// TwinCAT 3 PLC project TwinCAT_OpenFramework_FileSystem
// Title: TwinCAT Open Framework File System
// Company: Oleksandr Tiutyk FOP
// Author: Oleksandr Tiutyk
// ProjectVersion: 1.0.13.0
// Description: TwinCAT.OpenFramework classes to work with files and directories
// ProgramVersion: 3.1.4026.28
// libraries:
//   Tc2_System, * (Beckhoff Automation GmbH)
//   Tc2_Utilities, * (Beckhoff Automation GmbH)
//   [TwinCAT Open Framework Core], * (Oleksandr Tiutyk FOP)
//   [TwinCAT Open Framework Tasks], * (Oleksandr Tiutyk FOP)
// project tree:
//   Exceptions/ IInvalidPathException.TcIO, InvalidPathException.TcPOU, IFileSystemException.TcIO, FileSystemException.TcPOU, FileSystemExceptions.TcPOU
//   Internal/ CurrentNamespace.TcPOU, NamespaceExtractor.TcPOU
//   / PathHelper.TcPOU
//   Tasks/Directory/ CreateDirectoryIfNotExists.TcPOU, CreateDirectory.TcPOU, RemoveEmptyDirectoryIfExists.TcPOU, RemoveEmptyDirectory.TcPOU, CheckDirectoryExists.TcPOU
//   Tasks/File/ DeleteFile.TcPOU, LoadFile.TcPOU, RenameFile.TcPOU
//   Tasks/File/FileContent/ FileContentManager.TcPOU, FileHandleResourceManager.TcPOU, FileHandleResource.TcPOU
//   Tasks/File/FileContent/Tasks/ CheckEndOfFile.TcPOU, FileContentTask.TcPOU, GetPositionInFile.TcPOU (not stored), IFileContentTask.TcIO, ReadBytesFromFile.TcPOU (not stored), ReadString255FromFile.TcPOU (not stored), SetPositionInFile.TcPOU, WriteBytesToFile.TcPOU, WriteString255ToFile.TcPOU (not stored)
//   Tasks/ IFileSystemTask.TcIO
//   Version/ Global_Version.TcGVL
// (motion and I/O tree: see PLC project twincat_openframework_core)
// real-time tasks:
//   TASK PlcTask: cycle T#10ms, priority 20, ADS port 350
//   TASK TestTask: cycle T#10ms, priority 1, ADS port 351
//   TASK RunnerTestTask: cycle T#10ms, priority 2, ADS port 354
//   TASK HowToTask: cycle T#10ms, priority 22, ADS port 353
// variable links:

// ---- Version/Global_Version.TcGVL
{attribute 'TcGenerated'}
{attribute 'no-analysis'}
{attribute 'linkalways'}
// This function has been automatically generated from the project information.
VAR_GLOBAL CONSTANT
	{attribute 'const_non_replaced'}
	stLibVersion_TwinCAT_Open_Framework_File_System : ST_LibVersion := (iMajor := 1, iMinor := 0, iBuild := 13, iRevision := 0, nFlags := 0, sVersion := '1.0.13.0');
END_VAR

// ---- Exceptions/IInvalidPathException.TcIO
(*
SPDX-FileCopyrightText: © 2026 Oleksandr Tiutyk <trofimich@gmail.com>
SPDX-License-Identifier: MIT
License: https://opensource.org/license/mit
*)

(*!
<summary>Exposes diagnostics for a rejected filesystem path.</summary>
<description>
Reports caller-detected path errors using the GeneralException lifetime and throw rules. The path is borrowed
during the call; errorMessage is copied by value.
</description>
*)
INTERFACE IInvalidPathException EXTENDS TOF_Core.IGeneralException

(*!
<summary>Raises an exception describing the rejected path and its reason.</summary>
<description>
Borrows path read-only for this call and copies errorMessage by value, limited to 255 characters. Retains
formatted diagnostic text, not the input reference. The caller detects the invalid path; this method does not
validate it.
</description>
*)
METHOD Throw
VAR_INPUT
	sourceNamespaceName : STRING;
	sourceClassName : STRING;
	sourcePOUName : STRING;
	sourcePosition : STRING;
END_VAR
VAR_IN_OUT CONSTANT
	path : STRING(255);
END_VAR
VAR_INPUT
	errorMessage : WSTRING(255);
END_VAR
END_METHOD

END_INTERFACE

// ---- Exceptions/IFileSystemException.TcIO
(*
SPDX-FileCopyrightText: © 2026 Oleksandr Tiutyk <trofimich@gmail.com>
SPDX-License-Identifier: MIT
License: https://opensource.org/license/mit
*)

(*!
<summary>Exposes diagnostics for a filesystem operation failure.</summary>
<description>
Reports caller-detected filesystem errors, such as ADS/OS errors, using the GeneralException lifetime and
throw rules. Message is borrowed read-only during the call; errorCode holds the operation failure code.
</description>
*)
INTERFACE IFileSystemException EXTENDS TOF_Core.IGeneralException

(*!
<summary>Raises an exception describing the filesystem failure.</summary>
<description>
Borrows message read-only for this call and records the numeric error code. Retains formatted diagnostic text.
The caller detects the filesystem error; this method propagates it.
</description>
<param name="sourceNamespaceName">Namespace of the caller.</param>
<param name="sourceClassName">Class name of the caller.</param>
<param name="sourcePOUName">POU name of the caller.</param>
<param name="sourcePosition">Source position of the caller.</param>
<param name="message">Diagnostic explanation.</param>
<param name="errorCode">Native/ADS error code, or 0 if unassigned.</param>
*)
METHOD Throw
VAR_INPUT
	sourceNamespaceName : STRING;
	sourceClassName : STRING;
	sourcePOUName : STRING;
	sourcePosition : STRING;
END_VAR
VAR_IN_OUT CONSTANT
	message : TOF_Core.ERROR_MESSAGE;
END_VAR
VAR_INPUT
	errorCode : UDINT := 0;
END_VAR
END_METHOD

END_INTERFACE

// ---- Tasks/File/FileContent/Tasks/IFileContentTask.TcIO
(*!
<summary>Defines a queued file operation that borrows a manager-owned resource.</summary>
<description>
A child must be READY and absent from every queue before binding. While queued, keep it alive and let the
queue drive its lifecycle. Binding and queue membership transfer no ownership. Implementations must keep
borrowed resource data read-only and complete pending I/O before permitting resource release. Keep the
resource owner alive throughout use. Removing a queue entry does not clear the binding.
</description>
*)
INTERFACE IFileContentTask EXTENDS IFileSystemTask

(*!
<summary>Provides the native handle associated with the file resource.</summary>
<description>
Use only during the current acquisition; the value alone is not an acquisition guard. Do not close it
independently or retain it across release. FileContentTask returns zero when unbound.
</description>
*)
{attribute 'monitoring' := 'call'}
PROPERTY FileHandle : UINT
GET
END_GET
END_PROPERTY

(*!
<summary>Provides a copy of the path from the borrowed file resource.</summary>
<description>
The resource owner must remain alive during access. FileContentTask returns an empty string when unbound. The
path is configuration, not proof of acquisition or file existence.
</description>
*)
{attribute 'monitoring' := 'call'}
PROPERTY FINAL FilePath : Tc2_System.T_MaxString
GET
END_GET
END_PROPERTY

(*!
<summary>Bind, replace or clear a borrowed resource only in READY; otherwise throw.</summary>
<description>
An invalid reference clears the binding. Reset a STOPPED task before rebinding. The caller must first remove
the task from any queue; READY alone does not mean it is unqueued. The resource owner must outlive its use by
this task. FileContentTask clears binding on Reset from STOPPED, but its READY Reset is a no-op; a removed
READY child needs explicit clearing or rebinding.
</description>
*)

METHOD SetFileHandleResource
VAR_INPUT
	fileHandleResource : REFERENCE TO FileHandleResource;
END_VAR
END_METHOD

END_INTERFACE

// ---- Tasks/IFileSystemTask.TcIO
(*!
<summary>Provides task execution with a configured file-system target and operation timeout.</summary>
<description>
Before online change, the application must stop submitting new work and keep advancing each running task
through completion and cleanup. Keep its configuration, borrowed objects and buffers alive until then. Drive
queued children only through their owning queue. File-content tasks also require their resource owner to
finish release; a stopped child alone does not close its file. Online change with pending native operations or
retained open resources is unsupported. This is an application precondition, not an automatic online-change
guard. Completed best-effort cleanup does not certify physical resource release after a native close or
enumeration-abort failure.
</description>
*)
INTERFACE IFileSystemTask EXTENDS TOF_Tasks.ITask

(*!
<summary>Selects the ADS target for the native filesystem operation.</summary>
<description>
Configure before execution and keep stable through stopping. File-content tasks obtain the effective target
from their bound resource; assigning this property does not retarget an acquired file.
</description>
*)
{attribute 'monitoring' := 'call'}
PROPERTY AmsNetId : Tc2_System.T_AmsNetID
GET
END_GET
SET
END_SET
END_PROPERTY

(*!
<summary>Configures the timeout passed to native operation requests.</summary>
<description>
Implementations apply this value to their native requests. Configure before execution and keep stable through
stopping; it is not a deadline for the entire task lifecycle.
</description>
*)
{attribute 'monitoring' := 'call'}
PROPERTY Timeout : TIME
GET
END_GET
SET
END_SET
END_PROPERTY

END_INTERFACE

// ---- Exceptions/InvalidPathException.TcPOU
(*
SPDX-FileCopyrightText: © 2026 Oleksandr Tiutyk <trofimich@gmail.com>
SPDX-License-Identifier: MIT
License: https://opensource.org/license/mit
*)

(*!
<summary>Reports a rejected filesystem path and its diagnostic explanation.</summary>
<description>
Reports caller-detected path errors using the GeneralException lifetime and throw rules. The path is borrowed
during the call; errorMessage is copied by value. Dynamic copies are explicitly registered by Clone after
construction; plain __NEW does not transfer ownership to the task manager.
</description>
*)

{attribute 'enable_dynamic_creation'}
{attribute 'no_explicit_call' := 'do not call this function block directly'}
FUNCTION_BLOCK InvalidPathException EXTENDS TOF_Core.GeneralException IMPLEMENTS IInvalidPathException
VAR_STAT
	//! <summary>Class name shared by all instances of this function block.</summary>
	{attribute 'hide'} 
	_ClassName : STRING := __POUNAME();
END_VAR

(*!
<summary>Provides the concrete type name used in diagnostics.</summary>
<description>
Returns borrowed read-only metadata; keep the instance alive and do not modify the referenced string.
Reading does not allocate memory, initialize resources or transfer ownership.
</description>
*)
{attribute 'monitoring' := 'call'}
PROPERTY ClassName : REFERENCE TO STRING
GET
ClassName REF= _ClassName;
END_GET
END_PROPERTY

(*!
<summary>Creates a task-owned copy of this exception and its diagnostic payload.</summary>
<description>
Registers the newly constructed instance before copying payload, outside FB_init. Registration failure
releases the unregistered instance and raises a terminal error; copy failure leaves the registered instance
owned by the task manager for cleanup. Custom overrides must follow the same ownership sequence. The returned
reference is borrowed until task cleanup and must not be deleted by the caller.
</description>
*)
METHOD Clone : TOF_Core.IObject
VAR
	exceptionClone : POINTER TO InvalidPathException;
END_VAR
exceptionClone := __NEW(InvalidPathException);

IF exceptionClone = 0 THEN
	TOF_Core.DynamicMemoryManager.RaiseAllocationFailure();
END_IF

TOF_Core.DynamicMemoryManager.RegisterAutoDisposedObject(autoDisposedObject := exceptionClone^);

exceptionClone^.CopyGeneralFields(sourceException := THIS^);

Clone := exceptionClone^;
END_METHOD

(*!
<summary>Provides the library namespace used in diagnostics.</summary>
<description>Returns borrowed read-only namespace storage; do not modify the referenced string.</description>
*)
{attribute 'monitoring' := 'call'}
PROPERTY NamespaceName : REFERENCE TO STRING
GET
NamespaceName REF= CurrentNamespace.Name;
END_GET
END_PROPERTY

(*!
<summary>Reports the size of this concrete instance in bytes.</summary>
*)
{attribute 'monitoring' := 'call'}
PROPERTY SelfSize : ULINT
GET
SelfSize := XSIZEOF(THIS^);
END_GET
END_PROPERTY

(*!
<summary>Raises an exception describing the rejected path and its reason.</summary>
<description>
Borrows path read-only for this call and copies errorMessage by value, limited to 255 characters. Formats
diagnostic text without heap allocation during message preparation; does not retain the input reference. The
caller detects the invalid path; this method does not validate it.
</description>
*)
METHOD Throw
VAR_INPUT
	sourceNamespaceName : STRING;
	sourceClassName : STRING;
	sourcePOUName : STRING;
	sourcePosition : STRING;
END_VAR
VAR_IN_OUT CONSTANT
	path : STRING(255);
END_VAR
VAR_INPUT
	errorMessage : WSTRING(255);
END_VAR
VAR
	message : TOF_Core.ERROR_MESSAGE;
END_VAR
TOF_Core.WideStrings.Append255(
	message,
	"Invalid path ",
	TO_WSTRING('$22'),
	TO_WSTRING(path),
	TO_WSTRING('$22: '),
	errorMessage);

InternalThrow(
	sourceNamespaceName := sourceNamespaceName,
	sourceClassName := sourceClassName,
	sourcePOUName := sourcePOUName,
	sourcePosition := sourcePosition,
	message := message,
	errorCode := 0,
	innerException := 0
);
END_METHOD

END_FUNCTION_BLOCK

// ---- Internal/CurrentNamespace.TcPOU
(*
SPDX-FileCopyrightText: © 2026 Oleksandr Tiutyk <trofimich@gmail.com>
SPDX-License-Identifier: MIT
License: https://opensource.org/license/mit
*)

(*!
<summary>Owns the namespace storage shared by FileSystem diagnostic metadata.</summary>
*)

{attribute 'no_explicit_call' := 'do not call this POU directly'}
PROGRAM INTERNAL CurrentNamespace
VAR
	{attribute 'hide'} 
	_NamespaceExtractor : NamespaceExtractor;
END_VAR

(*!
<summary>Provides the compiler-initialized namespace string for this library.</summary>
<description>Returns borrowed read-only storage owned by the internal namespace extractor.</description>
*)
{attribute 'monitoring' := 'call'}
PROPERTY Name : REFERENCE TO STRING
GET
Name REF= _NamespaceExtractor.CurrentNamespace;
END_GET
END_PROPERTY

END_PROGRAM

// ---- Internal/NamespaceExtractor.TcPOU
(*
SPDX-FileCopyrightText: © 2026 Oleksandr Tiutyk <trofimich@gmail.com>
SPDX-License-Identifier: MIT
License: https://opensource.org/license/mit
*)

(*!
<summary>Receives the library namespace through compiler initialization.</summary>
<description>
CurrentNamespace is metadata storage; callers borrow it read-only through CurrentNamespace.Name.
</description>
*)

FUNCTION_BLOCK INTERNAL NamespaceExtractor
VAR_OUTPUT
	{attribute 'init_namespace'} 
	CurrentNamespace : STRING; 	
END_VAR

END_FUNCTION_BLOCK

// ---- Exceptions/FileSystemException.TcPOU
(*
SPDX-FileCopyrightText: © 2026 Oleksandr Tiutyk <trofimich@gmail.com>
SPDX-License-Identifier: MIT
License: https://opensource.org/license/mit
*)

(*!
<summary>Reports an error occurring during filesystem operations.</summary>
<description>
Reports caller-detected filesystem failures using the GeneralException lifetime and throw rules. Message is
borrowed read-only during the call; errorCode stores the native/ADS error identifier. Dynamic instances and
clones belong to DynamicMemoryManager until task cleanup. Plain __NEW does not transfer ownership to the task
manager.
</description>
*)

{attribute 'enable_dynamic_creation'}
{attribute 'no_explicit_call' := 'do not call this function block directly'}
FUNCTION_BLOCK FileSystemException EXTENDS TOF_Core.GeneralException IMPLEMENTS IFileSystemException
VAR_STAT
	{attribute 'hide'} 
	_ClassName : STRING := __POUNAME();
END_VAR

(*!
<summary>Provides the concrete type name used in diagnostics.</summary>
<description>
Returns borrowed read-only metadata; keep the instance alive and do not modify the referenced string.
Reading does not allocate memory, initialize resources or transfer ownership.
</description>
*)
{attribute 'monitoring' := 'call'}
PROPERTY ClassName : REFERENCE TO STRING
GET
ClassName REF= _ClassName;
END_GET
END_PROPERTY

(*!
<summary>Creates a task-owned copy of this exception and its diagnostic payload.</summary>
<description>
Registers the newly constructed instance before copying payload, outside FB_init. Registration failure
releases the unregistered instance and raises a terminal error; copy failure leaves the registered instance
owned by the task manager for cleanup. Custom overrides must follow the same ownership sequence. The returned
reference is borrowed until task cleanup and must not be deleted by the caller.
</description>
*)
METHOD Clone : TOF_Core.IObject
VAR
	exceptionClone : POINTER TO FileSystemException;
END_VAR
exceptionClone := __NEW(FileSystemException);

IF exceptionClone = 0 THEN
	TOF_Core.DynamicMemoryManager.RaiseAllocationFailure();
END_IF

TOF_Core.DynamicMemoryManager.RegisterAutoDisposedObject(autoDisposedObject := exceptionClone^);

exceptionClone^.CopyGeneralFields(sourceException := THIS^);

Clone := exceptionClone^;
END_METHOD

(*!
<summary>Provides the library namespace used in diagnostics.</summary>
<description>Returns borrowed read-only namespace storage; do not modify the referenced string.</description>
*)
{attribute 'monitoring' := 'call'}
PROPERTY NamespaceName : REFERENCE TO STRING
GET
NamespaceName REF= CurrentNamespace.Name;
END_GET
END_PROPERTY

(*!
<summary>Reports the size of this concrete instance in bytes.</summary>
*)
{attribute 'monitoring' := 'call'}
PROPERTY SelfSize : ULINT
GET
SelfSize := XSIZEOF(THIS^);
END_GET
END_PROPERTY

(*!
<summary>Raises a filesystem exception with the supplied message and error code.</summary>
<description>
Borrows message read-only for this call and records the numeric error code. Formats diagnostic text without
heap allocation during message preparation; does not retain the input reference. The caller detects the
filesystem error; this method propagates it.
</description>
<param name="sourceNamespaceName">Namespace of the caller.</param>
<param name="sourceClassName">Class name of the caller.</param>
<param name="sourcePOUName">POU name of the caller.</param>
<param name="sourcePosition">Source position of the caller.</param>
<param name="message">Diagnostic explanation.</param>
<param name="errorCode">Native/ADS error code, or 0 if unassigned.</param>
*)
METHOD Throw
VAR_INPUT
	sourceNamespaceName : STRING;
	sourceClassName : STRING;
	sourcePOUName : STRING;
	sourcePosition : STRING;
END_VAR
VAR_IN_OUT CONSTANT
	message : TOF_Core.ERROR_MESSAGE;
END_VAR
VAR_INPUT
	errorCode : UDINT := 0;
END_VAR
InternalThrow(
	sourceNamespaceName := sourceNamespaceName,
	sourceClassName := sourceClassName,
	sourcePOUName := sourcePOUName,
	sourcePosition := sourcePosition,
	message := message,
	errorCode := errorCode,
	innerException := 0
);
END_METHOD

END_FUNCTION_BLOCK

// ---- Exceptions/FileSystemExceptions.TcPOU
(*
SPDX-FileCopyrightText: © 2026 Oleksandr Tiutyk <trofimich@gmail.com>
SPDX-License-Identifier: MIT
License: https://opensource.org/license/mit
*)

(*!
<summary>Provides static helper methods for throwing FileSystem-specific exceptions.</summary>
<description>
Constructs stack-local template exceptions, formats diagnostics without heap allocation and propagates them
through ExceptionManager.
</description>
*)

PROGRAM FileSystemExceptions
VAR
	{attribute 'hide'} 
	_ClassName : STRING := __POUNAME();
END_VAR

//! <summary>Borrows the concrete class name for the lifetime of this instance; callers must not modify it.</summary>
{attribute 'monitoring' := 'call'}
PROPERTY ClassName : REFERENCE TO STRING
GET
ClassName REF= _ClassName;
END_GET
END_PROPERTY

//! <summary>Borrows the compiler-initialized namespace; callers must not modify the returned reference.</summary>
{attribute 'monitoring' := 'call'}
PROPERTY NamespaceName : REFERENCE TO STRING
GET
NamespaceName REF= CurrentNamespace.Name;
END_GET
END_PROPERTY

(*!
<summary>Raises a FileSystemException without requiring a caller-owned exception variable.</summary>
<description>Constructs a temporary stack template and delegates to FileSystemException.Throw.</description>
<param name="sourceNamespaceName">Namespace of the caller.</param>
<param name="sourceClassName">Class name of the caller.</param>
<param name="sourcePOUName">POU name of the caller.</param>
<param name="sourcePosition">Source position of the caller.</param>
<param name="message">Diagnostic explanation.</param>
<param name="errorCode">Native/ADS error code, or 0 if unassigned.</param>
*)
METHOD ThrowFileSystem
VAR_INPUT
	sourceNamespaceName : STRING;
	sourceClassName : STRING;
	sourcePOUName : STRING;
	sourcePosition : STRING;
END_VAR
VAR_IN_OUT CONSTANT
	message : TOF_Core.ERROR_MESSAGE;
END_VAR
VAR_INPUT
	errorCode : UDINT := 0;
END_VAR
VAR
	exception : FileSystemException;
END_VAR
exception.Throw(
	sourceNamespaceName := sourceNamespaceName,
	sourceClassName := sourceClassName,
	sourcePOUName := sourcePOUName,
	sourcePosition := sourcePosition,
	message := message,
	errorCode := errorCode
);
END_METHOD

(*!
<summary>Raises an InvalidPathException without requiring a caller-owned exception variable.</summary>
<description>Constructs a temporary stack template and delegates to InvalidPathException.Throw.</description>
<param name="sourceNamespaceName">Namespace of the caller.</param>
<param name="sourceClassName">Class name of the caller.</param>
<param name="sourcePOUName">POU name of the caller.</param>
<param name="sourcePosition">Source position of the caller.</param>
<param name="path">Rejected filesystem path.</param>
<param name="errorMessage">Diagnostic explanation.</param>
*)
METHOD ThrowInvalidPath
VAR_INPUT
	sourceNamespaceName : STRING;
	sourceClassName : STRING;
	sourcePOUName : STRING;
	sourcePosition : STRING;
END_VAR
VAR_IN_OUT CONSTANT
	path : STRING(255);
END_VAR
VAR_INPUT
	errorMessage : WSTRING(255);
END_VAR
VAR
	exception : InvalidPathException;
END_VAR
exception.Throw(
	sourceNamespaceName := sourceNamespaceName,
	sourceClassName := sourceClassName,
	sourcePOUName := sourcePOUName,
	sourcePosition := sourcePosition,
	path := path,
	errorMessage := errorMessage
);
END_METHOD

END_PROGRAM

// ---- PathHelper.TcPOU
(*
SPDX-FileCopyrightText: © 2026 Oleksandr Tiutyk <trofimich@gmail.com>
SPDX-License-Identifier: MIT
License: https://opensource.org/license/mit
*)

(*!
<summary>Provides lexical checks for directory and file path strings.</summary>
<description>
These checks perform no filesystem I/O, normalization or access checks. Passing does not certify acceptance by
a native service or target filesystem. The current filter is not a complete Windows, UNC or platform-specific
path validator; it does not validate reserved names or dot components. Callers must separately satisfy the
path requirements of the actual operation and target.
</description>
*)

{attribute 'no_explicit_call' := 'do not call this function block directly'}
PROGRAM PathHelper
VAR CONSTANT
	//! <summary>Drive-letter, colon and separator occupy the first three bytes of an absolute drive prefix.</summary>
	_DrivePrefixLength : UDINT := 3;
	//! <summary>Zero-based index of the colon immediately following a drive letter.</summary>
	_DriveColonIndex : UDINT := 1;
	//! <summary>Zero-based index of the separator following the drive colon.</summary>
	_DriveSeparatorIndex : UDINT := 2;
	//! <summary>Last index allowed in the initial separator pair before repeated separators are rejected.</summary>
	_LeadingSeparatorPairLastIndex : UDINT := 1;
END_VAR
VAR
	{attribute 'hide'} 
	_ClassName : STRING := __POUNAME();
END_VAR

//! <summary>Borrows the concrete class name for the lifetime of this instance; callers must not modify it.</summary>
{attribute 'monitoring' := 'call'}
PROPERTY ClassName : REFERENCE TO STRING
GET
ClassName REF= _ClassName;
END_GET
END_PROPERTY

(*!
<summary>Checks the lexical form of a directory path without accessing the filesystem.</summary>
<description>
Rejects an empty path, bytes below ASCII space, characters from the current forbidden set and repeated
slash/backslash separators beyond the leading pair. A colon is accepted only immediately after an ASCII drive
letter and before a separator. Relative paths and a trailing separator are not rejected solely for being
relative or trailing. Leading separator pairs are permitted lexically, but UNC server/share structure is not
checked and native network-path support is not implied. Reserved names, dot components and trailing
dots/spaces are not validated. TRUE means only that this filter passed; errorMessage is meaningful on FALSE.
Input is borrowed only for the call.
</description>
<param name="directoryPath">Directory path to inspect without modifying or retaining it.</param>
<param name="errorMessage">Reason for the first rejected condition.</param>
*)
METHOD IsValidDirectoryPath : BOOL
VAR_IN_OUT CONSTANT
	directoryPath : Tc2_System.T_MaxString;
END_VAR
VAR_OUTPUT
	errorMessage : WSTRING(255);
END_VAR
VAR
	i, j : UDINT;
	stringLength : UDINT;
	character : BYTE;

	(* Current lexical exclusions, not an OS-wide list. Caret is an existing library restriction;
	   the drive-letter exception below handles the only accepted colon position. *)
	invalidChars : STRING(8) := '<>"|?*^:';
END_VAR
stringLength := TOF_Core.Strings.GetLength(value := directoryPath);

IF stringLength = TOF_Core.UnsignedInt32.ZERO THEN
	errorMessage := "Path is empty";
	RETURN;
END_IF

FOR i := 0 TO stringLength - 1 DO
	character := directoryPath[i];

	(* A colon is allowed only in an absolute ASCII drive prefix. *)
	IF i = _DriveColonIndex AND_THEN character = Tc2_System.F_ToASC(str := ':') THEN

		IF stringLength >= _DrivePrefixLength
			AND_THEN (
				directoryPath[_DriveSeparatorIndex] = Tc2_System.F_ToASC(str := '\')
				OR_ELSE directoryPath[_DriveSeparatorIndex] = Tc2_System.F_ToASC(str := '/')
			)
			AND_THEN (
				(directoryPath[0] >= Tc2_System.F_ToASC(str := 'A')
					AND_THEN directoryPath[0] <= Tc2_System.F_ToASC(str := 'Z'))
				OR_ELSE (directoryPath[0] >= Tc2_System.F_ToASC(str := 'a')
					AND_THEN directoryPath[0] <= Tc2_System.F_ToASC(str := 'z'))
			)
		THEN
			CONTINUE;
		END_IF

	END_IF

	FOR j := 0 TO TOF_Core.Strings.GetLength(value := invalidChars) - 1 DO

		IF character = invalidChars[j] THEN
			errorMessage := TOF_Core.WideStrings.Concat255(
				"The forbidden character '",
				TO_WSTRING(Tc2_System.F_ToCHR(c := character)),
				"' at position ",
				TO_WSTRING(i + 1)
			);
			RETURN;
		END_IF

	END_FOR

	IF character < TOF_Core.Strings.ASCII_SPACE THEN
		errorMessage := TOF_Core.WideStrings.Concat255(
			"The forbidden character with code ",
			TO_WSTRING(character),
			" at position ",
			TO_WSTRING(i + 1)
		);
		RETURN;
	END_IF

	IF i > _LeadingSeparatorPairLastIndex
		AND_THEN (character = Tc2_System.F_ToASC(str := '\') OR_ELSE character = Tc2_System.F_ToASC(str := '/'))
		AND_THEN (
			directoryPath[i - 1] = Tc2_System.F_ToASC(str := '\')
			OR_ELSE directoryPath[i - 1] = Tc2_System.F_ToASC(str := '/')
		)
	THEN
		errorMessage := TOF_Core.WideStrings.Concat255("Several slashes one by one at position ", TO_WSTRING(i + 1));
		RETURN;
	END_IF

END_FOR

IsValidDirectoryPath := TRUE;
END_METHOD

(*!
<summary>Checks the lexical form of a file path and rejects a trailing separator.</summary>
<description>
Borrows the path only for this call. Returns FALSE with errorMessage for an empty path, a forbidden character,
repeated separators beyond the leading pair, or a final slash or backslash. A drive-letter colon is allowed
only before a slash or backslash. TRUE means the lexical checks passed; it does not establish file existence,
access rights or acceptance by the target filesystem. No filesystem I/O is performed. Relative paths are not
rejected solely for being relative. Leading separator pairs do not establish a valid UNC path; reserved names,
dot components and trailing dots/spaces are not validated. errorMessage is meaningful only when FALSE is
returned.
</description>
<param name="filePath">File path to inspect without modifying or retaining it.</param>
<param name="errorMessage">Receives the reason for the first rejected condition.</param>
*)
METHOD IsValidFilePath : BOOL
VAR_IN_OUT CONSTANT
	filePath : Tc2_System.T_MaxString;
END_VAR
VAR_OUTPUT
	errorMessage : WSTRING(255);
END_VAR
VAR
	i, j : UDINT;
	stringLength : UDINT;
	character : BYTE;

	(* Current lexical exclusions, not an OS-wide list. Caret is an existing library restriction;
	   the drive-letter exception below handles the only accepted colon position. *)
	invalidChars : STRING(8) := '<>"|?*^:';
END_VAR
stringLength := TOF_Core.Strings.GetLength(value := filePath);

IF stringLength = TOF_Core.UnsignedInt32.ZERO THEN
	errorMessage := "Path is empty";
	RETURN;
END_IF

FOR i := 0 TO stringLength - 1 DO
	character := filePath[i];

	(* A colon is allowed only in an absolute ASCII drive prefix. *)
	IF i = _DriveColonIndex AND_THEN character = Tc2_System.F_ToASC(str := ':') THEN

		IF stringLength >= _DrivePrefixLength
			AND_THEN (
				filePath[_DriveSeparatorIndex] = Tc2_System.F_ToASC(str := '\')
				OR_ELSE filePath[_DriveSeparatorIndex] = Tc2_System.F_ToASC(str := '/')
			)
			AND_THEN (
				(filePath[0] >= Tc2_System.F_ToASC(str := 'A')
					AND_THEN filePath[0] <= Tc2_System.F_ToASC(str := 'Z'))
				OR_ELSE (filePath[0] >= Tc2_System.F_ToASC(str := 'a')
					AND_THEN filePath[0] <= Tc2_System.F_ToASC(str := 'z'))
			)
		THEN
			CONTINUE;
		END_IF

	END_IF

	FOR j := 0 TO TOF_Core.Strings.GetLength(value := invalidChars) - 1 DO

		IF character = invalidChars[j] THEN
			errorMessage := TOF_Core.WideStrings.Concat255(
				"The forbidden character '",
				TO_WSTRING(Tc2_System.F_ToCHR(c := character)),
				"' at position ",
				TO_WSTRING(i + 1)
			);
			RETURN;
		END_IF

	END_FOR

	IF character < TOF_Core.Strings.ASCII_SPACE THEN
		errorMessage := TOF_Core.WideStrings.Concat255(
			"The forbidden character with code ",
			TO_WSTRING(character),
			" at position ",
			TO_WSTRING(i + 1)
		);
		RETURN;
	END_IF

	IF i > _LeadingSeparatorPairLastIndex
		AND_THEN (character = Tc2_System.F_ToASC(str := '\') OR_ELSE character = Tc2_System.F_ToASC(str := '/'))
		AND_THEN (
			filePath[i - 1] = Tc2_System.F_ToASC(str := '\')
			OR_ELSE filePath[i - 1] = Tc2_System.F_ToASC(str := '/')
		)
	THEN
		errorMessage := TOF_Core.WideStrings.Concat255("Several slashes one by one at position ", TO_WSTRING(i + 1));
		RETURN;
	END_IF

	IF i = stringLength - 1
		AND_THEN (character = Tc2_System.F_ToASC(str := '\') OR_ELSE character = Tc2_System.F_ToASC(str := '/'))
	THEN
		errorMessage := "Slash at the end of the path";
		RETURN;
	END_IF

END_FOR

IsValidFilePath := TRUE;
END_METHOD

//! <summary>Borrows the compiler-initialized namespace; callers must not modify the returned reference.</summary>
{attribute 'monitoring' := 'call'}
PROPERTY NamespaceName : REFERENCE TO STRING
GET
NamespaceName REF= CurrentNamespace.Name;
END_GET
END_PROPERTY

END_PROGRAM

// ---- Tasks/Directory/CreateDirectoryIfNotExists.TcPOU
(*
SPDX-FileCopyrightText: © 2026 Oleksandr Tiutyk <trofimich@gmail.com>
SPDX-License-Identifier: MIT
License: https://opensource.org/license/mit
*)

(*!
<summary>Creates a filesystem directory when it is absent.</summary>
<description>
An existing directory completes after native enumeration has been closed. Pending search and create commands
finish before stopping. Diagnostic string inputs are borrowed only during the call; retained diagnostic text
is copied into owned storage. A found file produces FAILURE without starting create I/O; stopping closes the
enumeration before task completion. The existence check and subsequent filesystem change are separate,
non-atomic operations. Another actor may change the same path between them. Native errors from the subsequent
create/remove are reported as failure; this wrapper does not retry or reinterpret them as a successful race.
Coordinate access externally when other tasks or processes can modify the same path. Cancellation does not
roll back completed filesystem effects.
</description>
*)

{attribute 'no_explicit_call' := 'do not call this function block directly'}
FUNCTION_BLOCK CreateDirectoryIfNotExists EXTENDS TOF_Tasks.Task IMPLEMENTS IFileSystemTask
VAR_STAT
	//! <summary>Static type metadata available before the base task initializes its default name.</summary>
	{attribute 'hide'}
	_ClassName : STRING := __POUNAME();
END_VAR
VAR
	_DirectoryChecking : BOOL;

	_EnumFindFile : Tc2_Utilities.FB_EnumFindFileEntry;
	//! <summary>Records whether a search command may still own native enumeration resources.</summary>
	_EnumerationStarted : BOOL;
	//! <summary>Prevents repeating the abort command while its completion is pending.</summary>
	_EnumerationAbortIssued : BOOL;

    _CreateDirectory : Tc2_System.FB_CreateDir;
END_VAR

(*!
<summary>Selects the ADS target for the native filesystem operation.</summary>
<description>
Configure before Start and keep unchanged until STOPPED; the setter stores configuration without submitting
I/O.
</description>
*)
{attribute 'monitoring' := 'call'}
PROPERTY AmsNetId : Tc2_System.T_AmsNetID
GET
AmsNetId := _CreateDirectory.sNetId;
END_GET
SET
_CreateDirectory.sNetId := AmsNetId;
_EnumFindFile.sNetId := AmsNetId;
END_SET
END_PROPERTY

(*!
<summary>Provides the concrete type name used in diagnostics.</summary>
<description>
Returns borrowed read-only metadata; keep the instance alive and do not modify the referenced string.
Initialized static storage is ready during base Task.FB_init; this getter has no side effects or exceptions.
</description>
*)
{attribute 'monitoring' := 'call'}
PROPERTY ClassName : REFERENCE TO STRING
GET
ClassName REF= _ClassName;
END_GET
END_PROPERTY

(*!
<summary>Provides the copied directory path used by the operation and its existence check.</summary>
<description>
Configure before Start and keep unchanged until STOPPED. PathHelper applies its limited lexical filter before
native submission. Assignment does not perform I/O; Reset preserves the path.
</description>
*)
{attribute 'monitoring' := 'call'}
PROPERTY DirectoryPath : Tc2_System.T_MaxString
GET
DirectoryPath := _CreateDirectory.sPathName;
END_GET
SET
_CreateDirectory.sPathName := DirectoryPath;
_EnumFindFile.sPathName := DirectoryPath;
END_SET
END_PROPERTY

(*!
<summary>Provides the library namespace used in diagnostics.</summary>
<description>Returns borrowed read-only namespace storage; do not modify the referenced string.</description>
*)
{attribute 'monitoring' := 'call'}
PROPERTY NamespaceName : REFERENCE TO STRING
GET
NamespaceName REF= CurrentNamespace.Name;
END_GET
END_PROPERTY

(*!
<summary>Clears completed directory operations and per-run enumeration cleanup state.</summary>
<description>Called only after stopping has completed; it does not abandon pending native I/O.</description>
*)
METHOD PROTECTED OnReset
_EnumFindFile(bExecute := FALSE);
_CreateDirectory(bExecute := FALSE);

_DirectoryChecking := FALSE;
_EnumerationStarted := FALSE;
_EnumerationAbortIssued := FALSE;
END_METHOD

(*!
<summary>Checks for a directory and creates it only if absent.</summary>
<description>
Early discovery leaves native search cleanup to OnStopping. A missing directory begins a create request after
bEOE. Computed diagnostics are held in local buffers for the receiving call without dynamic string-builder
allocations. A found file returns ERROR with a diagnostic message and leaves enumeration cleanup to
OnStopping; no create request starts.
</description>
<param name="processingState">
BUSY while searching or creating; DONE when no create is needed or creation ends; ERROR when the path refers
to a file.
</param>
<param name="stopReasonMessage">
Receives diagnostics when the path refers to a file; native failures use exceptions.
</param>
*)
METHOD PROTECTED OnRunning
VAR_OUTPUT
	processingState : TOF_Tasks.TASK_PROCESSING_STATE;
END_VAR
VAR_IN_OUT
	stopReasonMessage : TOF_Core.ERROR_MESSAGE;
END_VAR
VAR
	formattedExceptionMessage : TOF_Core.ERROR_MESSAGE;
	pathErrorMessage : WSTRING(255);
END_VAR
IF NOT _EnumFindFile.bExecute THEN 
	IF TOF_Core.Strings.IsNullOrWhiteSpace(stringToCheck := _EnumFindFile.sPathName) THEN
		TOF_Core.Exceptions.ThrowDataMemberNotSpecified(
			sourceNamespaceName := NamespaceName,
			sourceClassName := ClassName,
			sourcePOUName := __POUNAME(),
			sourcePosition := __POSITION(),
			dataMemberName := 'DirectoryPath'
		);		
	END_IF
	
	IF NOT PathHelper.IsValidDirectoryPath(directoryPath := _EnumFindFile.sPathName, errorMessage => pathErrorMessage) THEN
		FileSystemExceptions.ThrowInvalidPath(
			sourceNamespaceName := NamespaceName,
			sourceClassName := ClassName,
			sourcePOUName := __POUNAME(),
			sourcePosition := __POSITION(),
			path := _EnumFindFile.sPathName,
			errorMessage := pathErrorMessage
		);
	END_IF
	
	_DirectoryChecking := TRUE;
	
	_EnumFindFile.eCmd := Tc2_Utilities.E_EnumCmdType.eEnumCmd_First;
END_IF

IF _DirectoryChecking THEN
	_EnumerationStarted := TRUE;
	_EnumFindFile(bExecute := TRUE);
	
	IF _EnumFindFile.bError THEN
		TOF_Core.WideStrings.Append255(
			formattedExceptionMessage,
			"Error while checking directory '",
			TO_WSTRING(_EnumFindFile.sPathName),
			"'");

		FileSystemExceptions.ThrowFileSystem(
			sourceNamespaceName := NamespaceName,
			sourceClassName := ClassName,
			sourcePOUName := __POUNAME(),
			sourcePosition := __POSITION(),
			message := formattedExceptionMessage,
			errorCode := _EnumFindFile.nErrId
		);
	ELSIF NOT _EnumFindFile.bBusy THEN	
		_DirectoryChecking := FALSE;
		
		IF NOT _EnumFindFile.bEOE THEN
			IF _EnumFindFile.stFindFile.fileAttributes.bDirectory THEN
				processingState := TOF_Tasks.TASK_PROCESSING_STATE.DONE;
			ELSE
				stopReasonMessage := TOF_Core.WideStrings.Concat255("Directory path refers to a file: ", TO_WSTRING(_EnumFindFile.sPathName));
				processingState := TOF_Tasks.TASK_PROCESSING_STATE.ERROR;
			END_IF
		END_IF
	END_IF
ELSE
	_CreateDirectory(bExecute := TRUE);
	
	IF _CreateDirectory.bError THEN
		TOF_Core.WideStrings.Append255(
			formattedExceptionMessage,
			"Error while creating directory '",
			TO_WSTRING(_CreateDirectory.sPathName),
			"'");

		FileSystemExceptions.ThrowFileSystem(
			sourceNamespaceName := NamespaceName,
			sourceClassName := ClassName,
			sourcePOUName := __POUNAME(),
			sourcePosition := __POSITION(),
			message := formattedExceptionMessage,
			errorCode := _CreateDirectory.nErrId
		);
	END_IF
	
	IF NOT _CreateDirectory.bBusy THEN
		processingState := TOF_Tasks.TASK_PROCESSING_STATE.DONE;
	END_IF	
END_IF
END_METHOD

(*!
<summary>Advances directory stop actions before reporting termination.</summary>
<description>
Used for every stop reason. Drains a pending search, then issues an abort with a rising bExecute edge if the
search ended before bEOE without error. Waits for abort and any pending create operation before termination;
no new ordinary create request starts. An abort error is logged once with its native code and path, without
retrying abort or replacing the task stop reason. Readiness means this cleanup attempt ended, not that server
resources were proven released. The log attempt is made after clearing pending enumeration state; logger
failure does not restart cleanup.
</description>
<param name="readyToRelease">TRUE when the directory FBs have finished their pending requests.</param>
*)
METHOD PROTECTED OnStopping
VAR_OUTPUT
	readyToRelease : BOOL;
END_VAR
VAR
	enumerationAbortMessage : WSTRING(255);
END_VAR
IF _EnumerationStarted THEN
	_EnumFindFile(bExecute := FALSE);

	IF NOT _EnumFindFile.bBusy THEN

		IF _EnumFindFile.bEOE OR_ELSE _EnumFindFile.bError THEN
			_EnumerationStarted := FALSE;

			(* End this attempt before reporting its error so logging cannot cause repeated aborts. *)

			IF _EnumerationAbortIssued AND_THEN _EnumFindFile.bError THEN
				enumerationAbortMessage := TOF_Core.WideStrings.Concat255(
					"Directory enumeration abort failed (native error code ",
					TO_WSTRING(_EnumFindFile.nErrId),
					"): ",
					TO_WSTRING(_EnumFindFile.sPathName)
				);
				TryLogDiagnosticMessage(
					message := enumerationAbortMessage,
					category := TOF_Core.LOG_CATEGORY.ERROR,
					topic1 := TO_WSTRING(__POUNAME())
				);
			END_IF

		ELSIF NOT _EnumerationAbortIssued THEN
			_EnumFindFile(bExecute := TRUE, eCmd := Tc2_Utilities.E_EnumCmdType.eEnumCmd_Abort);
			_EnumerationAbortIssued := TRUE;
		ELSE
			_EnumerationStarted := FALSE;
		END_IF

	END_IF

END_IF

_CreateDirectory(bExecute := FALSE);

readyToRelease := NOT _EnumerationStarted AND_THEN NOT _CreateDirectory.bBusy;
END_METHOD

(*!
<summary>Selects the native path context for the filesystem request.</summary>
<description>
Configure before Start and keep unchanged until STOPPED. It is passed to the native operation, not used as a
path-validity result. Reset preserves it. Target support includes the ePath enumeration input in
Tc2_Utilities 3.10.9.
</description>
*)
{attribute 'monitoring' := 'call'}
PROPERTY PathType : Tc2_System.E_OpenPath
GET
PathType := _CreateDirectory.ePath;
END_GET
SET
_CreateDirectory.ePath := PathType;
_EnumFindFile.ePath := PathType;
END_SET
END_PROPERTY

(*!
<summary>Reports the size of this concrete instance in bytes.</summary>
*)
{attribute 'monitoring' := 'call'}
PROPERTY SelfSize : ULINT
GET
SelfSize := XSIZEOF(THIS^);
END_GET
END_PROPERTY

(*!
<summary>Configures the timeout passed to native operation requests.</summary>
<description>
Set before Start and keep unchanged until STOPPED. Reset preserves this value. It is not an overall task
deadline or a guarantee of resource release after a timeout.
</description>
*)
{attribute 'monitoring' := 'call'}
PROPERTY Timeout : TIME
GET
Timeout := _CreateDirectory.tTimeout;
END_GET
SET
_CreateDirectory.tTimeout := Timeout;
_EnumFindFile.tTimeout := Timeout;
END_SET
END_PROPERTY

END_FUNCTION_BLOCK

// ---- Tasks/Directory/CreateDirectory.TcPOU
(*
SPDX-FileCopyrightText: © 2026 Oleksandr Tiutyk <trofimich@gmail.com>
SPDX-License-Identifier: MIT
License: https://opensource.org/license/mit
*)

(*!
<summary>Creates a filesystem directory through cyclic task execution.</summary>
<description>
Configure DirectoryPath, PathType, AmsNetId and Timeout before Start and keep them unchanged until STOPPED.
The path must be nonblank and pass PathHelper's limited lexical filter; native services determine whether the
requested operation is supported. This task does not perform an existence precheck or suppress native errors.
Invalid configuration and native errors use the base Task failure and cleanup path. Cancellation waits for
submitted I/O without rolling back completed filesystem changes. Reset clears the native request state and
preserves configuration. Use one owner task per instance.
</description>
*)

{attribute 'no_explicit_call' := 'do not call this function block directly'}
FUNCTION_BLOCK CreateDirectory EXTENDS TOF_Tasks.Task IMPLEMENTS IFileSystemTask
VAR_STAT
	//! <summary>Static type metadata available before the base task initializes its default name.</summary>
	{attribute 'hide'}
	_ClassName : STRING := __POUNAME();
END_VAR
VAR
    _CreateDirectory : Tc2_System.FB_CreateDir;
END_VAR

(*!
<summary>Selects the ADS target for the native filesystem operation.</summary>
<description>
Configure before Start and keep unchanged until STOPPED; the setter stores configuration without submitting
I/O.
</description>
*)
{attribute 'monitoring' := 'call'}
PROPERTY AmsNetId : Tc2_System.T_AmsNetID
GET
AmsNetId := _CreateDirectory.sNetId;
END_GET
SET
_CreateDirectory.sNetId := AmsNetId;
END_SET
END_PROPERTY

(*!
<summary>Provides the concrete type name used in diagnostics.</summary>
<description>
Returns borrowed read-only metadata; keep the instance alive and do not modify the referenced string.
Initialized static storage is ready during base Task.FB_init; this getter has no side effects or exceptions.
</description>
*)
{attribute 'monitoring' := 'call'}
PROPERTY ClassName : REFERENCE TO STRING
GET
ClassName REF= _ClassName;
END_GET
END_PROPERTY

{attribute 'monitoring' := 'call'}
(*!
<summary>Provides the copied path for the next directory operation.</summary>
<description>
Set before Start and keep unchanged until STOPPED. Checked by PathHelper before submission, then interpreted
by the native service using PathType. Assignment does not perform I/O; Reset preserves it.
</description>
*)
PROPERTY DirectoryPath : Tc2_System.T_MaxString
GET
DirectoryPath := _CreateDirectory.sPathName;
END_GET
SET
_CreateDirectory.sPathName := DirectoryPath;
END_SET
END_PROPERTY

(*!
<summary>Provides the library namespace used in diagnostics.</summary>
<description>Returns borrowed read-only namespace storage; do not modify the referenced string.</description>
*)
{attribute 'monitoring' := 'call'}
PROPERTY NamespaceName : REFERENCE TO STRING
GET
NamespaceName REF= CurrentNamespace.Name;
END_GET
END_PROPERTY

(*!
<summary>Resets the native request edge after the task has stopped.</summary>
<description>
Preserves configured inputs and does not undo completed filesystem effects. Pending I/O must finish during
stopping before this hook runs.
</description>
*)
METHOD PROTECTED OnReset
_CreateDirectory(bExecute := FALSE);
END_METHOD

(*!
<summary>Validates the configured path and advances the native directory-create request.</summary>
<description>
Computed diagnostic strings are held in local buffers for the duration of the receiving call without dynamic
string-builder allocations.
</description>
*)
METHOD PROTECTED OnRunning
VAR_OUTPUT
	processingState : TOF_Tasks.TASK_PROCESSING_STATE;
END_VAR
VAR_IN_OUT
	stopReasonMessage : TOF_Core.ERROR_MESSAGE;
END_VAR
VAR	
	pathErrorMessage : WSTRING(255);
	formattedExceptionMessage : TOF_Core.ERROR_MESSAGE;
END_VAR
IF NOT _CreateDirectory.bExecute THEN 
	IF TOF_Core.Strings.IsNullOrWhiteSpace(stringToCheck := _CreateDirectory.sPathName) THEN
		TOF_Core.Exceptions.ThrowDataMemberNotSpecified(
			sourceNamespaceName := NamespaceName,
			sourceClassName := ClassName,
			sourcePOUName := __POUNAME(),
			sourcePosition := __POSITION(),
			dataMemberName := 'DirectoryPath'
		);		
	END_IF
	
	IF NOT PathHelper.IsValidDirectoryPath(directoryPath := _CreateDirectory.sPathName, errorMessage => pathErrorMessage) THEN
		FileSystemExceptions.ThrowInvalidPath(
			sourceNamespaceName := NamespaceName,
			sourceClassName := ClassName,
			sourcePOUName := __POUNAME(),
			sourcePosition := __POSITION(),
			path := _CreateDirectory.sPathName,
			errorMessage := pathErrorMessage
		);
	END_IF
END_IF

_CreateDirectory(bExecute := TRUE);

IF _CreateDirectory.bError THEN
	TOF_Core.WideStrings.Append255(
		formattedExceptionMessage,
		"Error while creating directory '",
		TO_WSTRING(_CreateDirectory.sPathName),
		"'");

	FileSystemExceptions.ThrowFileSystem(
		sourceNamespaceName := NamespaceName,
		sourceClassName := ClassName,
		sourcePOUName := __POUNAME(),
		sourcePosition := __POSITION(),
		message := formattedExceptionMessage,
		errorCode := _CreateDirectory.nErrId
	);
ELSIF NOT _CreateDirectory.bBusy THEN
	processingState := TOF_Tasks.TASK_PROCESSING_STATE.DONE;
END_IF
END_METHOD

(*!
<summary>Waits for an already submitted operation before task termination.</summary>
<description>
Runs for every stop reason. Advances the pending FB with bExecute=FALSE without issuing another request.
Completion does not roll back side effects. Keep configuration and borrowed buffers valid until STOPPED.
</description>
<param name="readyToRelease">TRUE when the underlying FB is no longer busy.</param>
*)
METHOD PROTECTED OnStopping
VAR_OUTPUT
	readyToRelease : BOOL;
END_VAR
IF _CreateDirectory.bBusy THEN
	_CreateDirectory(bExecute := FALSE);
END_IF

readyToRelease := NOT _CreateDirectory.bBusy;
END_METHOD

(*!
<summary>Selects the native path context for the filesystem request.</summary>
<description>
Configure before Start and keep unchanged until STOPPED. It is passed to the native operation, not used as a
path-validity result. Reset preserves it.
</description>
*)
{attribute 'monitoring' := 'call'}
PROPERTY PathType : Tc2_System.E_OpenPath
GET
PathType := _CreateDirectory.ePath;
END_GET
SET
_CreateDirectory.ePath := PathType;
END_SET
END_PROPERTY

(*!
<summary>Reports the size of this concrete instance in bytes.</summary>
*)
{attribute 'monitoring' := 'call'}
PROPERTY SelfSize : ULINT
GET
SelfSize := XSIZEOF(THIS^);
END_GET
END_PROPERTY

(*!
<summary>Configures the timeout passed to native operation requests.</summary>
<description>
Set before Start and keep unchanged until STOPPED. Reset preserves this value. It is not an overall task
deadline or a guarantee of resource release after a timeout.
</description>
*)
{attribute 'monitoring' := 'call'}
PROPERTY Timeout : TIME
GET
Timeout := _CreateDirectory.tTimeout;
END_GET
SET
_CreateDirectory.tTimeout := Timeout;
END_SET
END_PROPERTY

END_FUNCTION_BLOCK

// ---- Tasks/Directory/RemoveEmptyDirectoryIfExists.TcPOU
(*
SPDX-FileCopyrightText: © 2026 Oleksandr Tiutyk <trofimich@gmail.com>
SPDX-License-Identifier: MIT
License: https://opensource.org/license/mit
*)

(*!
<summary>Removes an empty filesystem directory when it exists.</summary>
<description>
Closes native enumeration before starting removal when a directory is found. Pending search and remove
commands finish before stopping. Diagnostic string inputs are borrowed only during the call; retained
diagnostic text is copied into owned storage. A found file produces FAILURE without starting remove I/O;
stopping closes the enumeration before task completion. The existence check and subsequent filesystem change
are separate, non-atomic operations. Another actor may change the same path between them. Native errors from
the subsequent create/remove are reported as failure; this wrapper does not retry or reinterpret them as a
successful race. Coordinate access externally when other tasks or processes can modify the same path.
Cancellation does not roll back completed filesystem effects.
</description>
*)

{attribute 'no_explicit_call' := 'do not call this function block directly'}
FUNCTION_BLOCK RemoveEmptyDirectoryIfExists EXTENDS TOF_Tasks.Task IMPLEMENTS IFileSystemTask
VAR_STAT
	//! <summary>Static type metadata available before the base task initializes its default name.</summary>
	{attribute 'hide'}
	_ClassName : STRING := __POUNAME();
END_VAR
VAR
	_DirectoryChecking : BOOL;

	_EnumFindFile : Tc2_Utilities.FB_EnumFindFileEntry;
	//! <summary>Records whether a search command may still own native enumeration resources.</summary>
	_EnumerationStarted : BOOL;
	//! <summary>Prevents repeating the abort command while its completion is pending.</summary>
	_EnumerationAbortIssued : BOOL;

    _RemoveDirectory : Tc2_System.FB_RemoveDir;
	
	//! <summary>Latches a found directory for this run so removal cannot restart the search.</summary>
	_DirectoryFound : BOOL;
END_VAR

(*!
<summary>Completes an active directory search before deletion or task termination.</summary>
<description>
Deasserts bExecute while a search command is pending. After a nonterminal search result, issues one abort with
a fresh rising edge and waits for its completion. bEOE and native errors close the enumeration without an
explicit abort. FALSE means the caller must resume on a later Execute. An abort error is logged once with its
native code and path, without retrying abort or replacing the task stop reason. Readiness means this cleanup
attempt ended, not that server resources were proven released. The log attempt is made after clearing pending
enumeration state; logger failure does not restart cleanup.
</description>
*)
METHOD PRIVATE advanceEnumerationClosure : BOOL
VAR
	enumerationAbortMessage : WSTRING(255);
END_VAR
advanceEnumerationClosure := FALSE;

IF NOT _EnumerationStarted THEN
	advanceEnumerationClosure := TRUE;
	RETURN;
END_IF

_EnumFindFile(bExecute := FALSE);

IF _EnumFindFile.bBusy THEN
	RETURN;
END_IF

IF _EnumFindFile.bEOE OR_ELSE _EnumFindFile.bError THEN
	_EnumerationStarted := FALSE;

	(* End this attempt before reporting its error so logging cannot cause repeated aborts. *)
	IF _EnumerationAbortIssued AND_THEN _EnumFindFile.bError THEN
		enumerationAbortMessage := TOF_Core.WideStrings.Concat255(
			"Directory enumeration abort failed (native error code ",
			TO_WSTRING(_EnumFindFile.nErrId),
			"): ",
			TO_WSTRING(_EnumFindFile.sPathName)
		);
		TOF_Core.LogManager.TryLogMessage(
			message := enumerationAbortMessage,
			category := TOF_Core.LOG_CATEGORY.ERROR,
			topic1 := TO_WSTRING(__POUNAME())
		);
	END_IF

	advanceEnumerationClosure := TRUE;
	RETURN;
END_IF

IF NOT _EnumerationAbortIssued THEN
	_EnumFindFile(bExecute := TRUE, eCmd := Tc2_Utilities.E_EnumCmdType.eEnumCmd_Abort);
	_EnumerationAbortIssued := TRUE;
	RETURN;
END_IF

_EnumerationStarted := FALSE;
advanceEnumerationClosure := TRUE;
END_METHOD

(*!
<summary>Selects the ADS target for the native filesystem operation.</summary>
<description>
Configure before Start and keep unchanged until STOPPED; the setter stores configuration without submitting
I/O.
</description>
*)
{attribute 'monitoring' := 'call'}
PROPERTY AmsNetId : Tc2_System.T_AmsNetID
GET
AmsNetId := _RemoveDirectory.sNetId;
END_GET
SET
_RemoveDirectory.sNetId := AmsNetId;
_EnumFindFile.sNetId := AmsNetId;
END_SET
END_PROPERTY

(*!
<summary>Provides the concrete type name used in diagnostics.</summary>
<description>
Returns borrowed read-only metadata; keep the instance alive and do not modify the referenced string.
Initialized static storage is ready during base Task.FB_init; this getter has no side effects or exceptions.
</description>
*)
{attribute 'monitoring' := 'call'}
PROPERTY ClassName : REFERENCE TO STRING
GET
ClassName REF= _ClassName;
END_GET
END_PROPERTY

(*!
<summary>Provides the copied directory path used by the operation and its existence check.</summary>
<description>
Configure before Start and keep unchanged until STOPPED. PathHelper applies its limited lexical filter before
native submission. Assignment does not perform I/O; Reset preserves the path.
</description>
*)
{attribute 'monitoring' := 'call'}
PROPERTY DirectoryPath : Tc2_System.T_MaxString
GET
DirectoryPath := _RemoveDirectory.sPathName;
END_GET
SET
_RemoveDirectory.sPathName := DirectoryPath;
_EnumFindFile.sPathName := DirectoryPath;
END_SET
END_PROPERTY

(*!
<summary>Provides the library namespace used in diagnostics.</summary>
<description>Returns borrowed read-only namespace storage; do not modify the referenced string.</description>
*)
{attribute 'monitoring' := 'call'}
PROPERTY NamespaceName : REFERENCE TO STRING
GET
NamespaceName REF= CurrentNamespace.Name;
END_GET
END_PROPERTY

(*!
<summary>Clears completed directory operations and per-run enumeration cleanup state.</summary>
<description>Called only after stopping has completed; it does not abandon pending native I/O.</description>
*)
METHOD PROTECTED OnReset
_EnumFindFile(bExecute := FALSE);
_RemoveDirectory(bExecute := FALSE);

_DirectoryChecking := FALSE;
_DirectoryFound := FALSE;
_EnumerationStarted := FALSE;
_EnumerationAbortIssued := FALSE;
END_METHOD

(*!
<summary>Checks for a directory and removes it only after closing the search.</summary>
<description>
On early discovery, the search abort must complete before the remove FB is started. A missing directory
completes successfully. Computed diagnostics are held in local buffers for the receiving call without dynamic
string-builder allocations. A found file returns ERROR with a diagnostic message and leaves enumeration
cleanup to OnStopping; no remove request starts.
</description>
<param name="processingState">
BUSY while searching, closing the search or removing; DONE after completion; ERROR when the path refers to a
file.
</param>
<param name="stopReasonMessage">
Receives diagnostics when the path refers to a file; native failures use exceptions.
</param>
*)
METHOD PROTECTED OnRunning
VAR_OUTPUT
	processingState : TOF_Tasks.TASK_PROCESSING_STATE;
END_VAR
VAR_IN_OUT
	stopReasonMessage : TOF_Core.ERROR_MESSAGE;
END_VAR
VAR
	formattedExceptionMessage : TOF_Core.ERROR_MESSAGE;
	pathErrorMessage : WSTRING(255);
END_VAR
IF NOT _DirectoryChecking AND_THEN NOT _EnumerationStarted AND_THEN NOT _DirectoryFound
THEN
	IF TOF_Core.Strings.IsNullOrWhiteSpace(stringToCheck := _EnumFindFile.sPathName) THEN
		TOF_Core.Exceptions.ThrowDataMemberNotSpecified(
			sourceNamespaceName := NamespaceName,
			sourceClassName := ClassName,
			sourcePOUName := __POUNAME(),
			sourcePosition := __POSITION(),
			dataMemberName := 'DirectoryPath'
		);		
	END_IF
	
	IF NOT PathHelper.IsValidDirectoryPath(directoryPath := _EnumFindFile.sPathName, errorMessage => pathErrorMessage) THEN
		FileSystemExceptions.ThrowInvalidPath(
			sourceNamespaceName := NamespaceName,
			sourceClassName := ClassName,
			sourcePOUName := __POUNAME(),
			sourcePosition := __POSITION(),
			path := _EnumFindFile.sPathName,
			errorMessage := pathErrorMessage
		);
	END_IF
	
	_DirectoryChecking := TRUE;
	
	_EnumFindFile(bExecute := FALSE, eCmd := Tc2_Utilities.E_EnumCmdType.eEnumCmd_First);
	_RemoveDirectory(bExecute := FALSE);
END_IF

IF _DirectoryChecking THEN
	_EnumerationStarted := TRUE;
	_EnumFindFile(bExecute := TRUE);
	
	IF _EnumFindFile.bError THEN
		TOF_Core.WideStrings.Append255(
			formattedExceptionMessage,
			"Error while checking directory '",
			TO_WSTRING(_EnumFindFile.sPathName),
			"'");

		FileSystemExceptions.ThrowFileSystem(
			sourceNamespaceName := NamespaceName,
			sourceClassName := ClassName,
			sourcePOUName := __POUNAME(),
			sourcePosition := __POSITION(),
			message := formattedExceptionMessage,
			errorCode := _EnumFindFile.nErrId
		);
	ELSIF NOT _EnumFindFile.bBusy THEN	
		_DirectoryChecking := FALSE;
		
		IF NOT _EnumFindFile.bEOE THEN
			IF _EnumFindFile.stFindFile.fileAttributes.bDirectory THEN
				_DirectoryFound := TRUE;
			ELSE
				stopReasonMessage := TOF_Core.WideStrings.Concat255("Directory path refers to a file: ", TO_WSTRING(_EnumFindFile.sPathName));
				processingState := TOF_Tasks.TASK_PROCESSING_STATE.ERROR;
			END_IF
		ELSE
			processingState := TOF_Tasks.TASK_PROCESSING_STATE.DONE;
		END_IF
	END_IF
ELSE
	IF NOT advanceEnumerationClosure() THEN
		RETURN;
	END_IF

	_RemoveDirectory(bExecute := TRUE);
	
	IF _RemoveDirectory.bError THEN
		TOF_Core.WideStrings.Append255(
			formattedExceptionMessage,
			"Error while removing directory '",
			TO_WSTRING(_RemoveDirectory.sPathName),
			"'");

		FileSystemExceptions.ThrowFileSystem(
			sourceNamespaceName := NamespaceName,
			sourceClassName := ClassName,
			sourcePOUName := __POUNAME(),
			sourcePosition := __POSITION(),
			message := formattedExceptionMessage,
			errorCode := _RemoveDirectory.nErrId
		);
	END_IF
	
	IF NOT _RemoveDirectory.bBusy THEN
		processingState := TOF_Tasks.TASK_PROCESSING_STATE.DONE;
	END_IF	
END_IF
END_METHOD

(*!
<summary>Advances directory stop actions before reporting termination.</summary>
<description>
Used for every stop reason. Finishes any search command and its required abort, then waits for pending remove
I/O. A new remove request is never started here. Readiness reports native FB completion, not server rollback.
</description>
<param name="readyToRelease">TRUE when the directory FBs have finished their pending requests.</param>
*)
METHOD PROTECTED OnStopping
VAR_OUTPUT
	readyToRelease : BOOL;
END_VAR
readyToRelease := advanceEnumerationClosure();

_RemoveDirectory(bExecute := FALSE);

readyToRelease := readyToRelease AND_THEN NOT _RemoveDirectory.bBusy;
END_METHOD

(*!
<summary>Selects the native path context for the filesystem request.</summary>
<description>
Configure before Start and keep unchanged until STOPPED. It is passed to the native operation, not used as a
path-validity result. Reset preserves it. Target support includes the ePath enumeration input in
Tc2_Utilities 3.10.9.
</description>
*)
{attribute 'monitoring' := 'call'}
PROPERTY PathType : Tc2_System.E_OpenPath
GET
PathType := _RemoveDirectory.ePath;
END_GET
SET
_RemoveDirectory.ePath := PathType;
_EnumFindFile.ePath := PathType;
END_SET
END_PROPERTY

(*!
<summary>Reports the size of this concrete instance in bytes.</summary>
*)
{attribute 'monitoring' := 'call'}
PROPERTY SelfSize : ULINT
GET
SelfSize := XSIZEOF(THIS^);
END_GET
END_PROPERTY

(*!
<summary>Configures the timeout passed to native operation requests.</summary>
<description>
Set before Start and keep unchanged until STOPPED. Reset preserves this value. It is not an overall task
deadline or a guarantee of resource release after a timeout.
</description>
*)
{attribute 'monitoring' := 'call'}
PROPERTY Timeout : TIME
GET
Timeout := _RemoveDirectory.tTimeout;
END_GET
SET
_RemoveDirectory.tTimeout := Timeout;
_EnumFindFile.tTimeout := Timeout;
END_SET
END_PROPERTY

END_FUNCTION_BLOCK

// ---- Tasks/Directory/RemoveEmptyDirectory.TcPOU
(*
SPDX-FileCopyrightText: © 2026 Oleksandr Tiutyk <trofimich@gmail.com>
SPDX-License-Identifier: MIT
License: https://opensource.org/license/mit
*)

(*!
<summary>Removes an empty filesystem directory through cyclic task execution.</summary>
<description>
Configure DirectoryPath, PathType, AmsNetId and Timeout before Start and keep them unchanged until STOPPED.
The path must be nonblank and pass PathHelper's limited lexical filter; native services determine whether the
requested operation is supported. This task does not perform an existence precheck or suppress native errors.
Invalid configuration and native errors use the base Task failure and cleanup path. Cancellation waits for
submitted I/O without rolling back completed filesystem changes. Reset clears the native request state and
preserves configuration. Use one owner task per instance.
</description>
*)

{attribute 'no_explicit_call' := 'do not call this function block directly'}
FUNCTION_BLOCK RemoveEmptyDirectory EXTENDS TOF_Tasks.Task IMPLEMENTS IFileSystemTask
VAR_STAT
	//! <summary>Static type metadata available before the base task initializes its default name.</summary>
	{attribute 'hide'}
	_ClassName : STRING := __POUNAME();
END_VAR
VAR
    _RemoveDirectory : Tc2_System.FB_RemoveDir;	
END_VAR

(*!
<summary>Selects the ADS target for the native filesystem operation.</summary>
<description>
Configure before Start and keep unchanged until STOPPED; the setter stores configuration without submitting
I/O.
</description>
*)
{attribute 'monitoring' := 'call'}
PROPERTY AmsNetId : Tc2_System.T_AmsNetID
GET
AmsNetId := _RemoveDirectory.sNetId;
END_GET
SET
_RemoveDirectory.sNetId := AmsNetId;
END_SET
END_PROPERTY

(*!
<summary>Provides the concrete type name used in diagnostics.</summary>
<description>
Returns borrowed read-only metadata; keep the instance alive and do not modify the referenced string.
Initialized static storage is ready during base Task.FB_init; this getter has no side effects or exceptions.
</description>
*)
{attribute 'monitoring' := 'call'}
PROPERTY ClassName : REFERENCE TO STRING
GET
ClassName REF= _ClassName;
END_GET
END_PROPERTY

{attribute 'monitoring' := 'call'}
(*!
<summary>Provides the copied path for the next directory operation.</summary>
<description>
Set before Start and keep unchanged until STOPPED. Checked by PathHelper before submission, then interpreted
by the native service using PathType. Assignment does not perform I/O; Reset preserves it.
</description>
*)
PROPERTY DirectoryPath : Tc2_System.T_MaxString
GET
DirectoryPath := _RemoveDirectory.sPathName;
END_GET
SET
_RemoveDirectory.sPathName := DirectoryPath;
END_SET
END_PROPERTY

(*!
<summary>Provides the library namespace used in diagnostics.</summary>
<description>Returns borrowed read-only namespace storage; do not modify the referenced string.</description>
*)
{attribute 'monitoring' := 'call'}
PROPERTY NamespaceName : REFERENCE TO STRING
GET
NamespaceName REF= CurrentNamespace.Name;
END_GET
END_PROPERTY

(*!
<summary>Resets the native request edge after the task has stopped.</summary>
<description>
Preserves configured inputs and does not undo completed filesystem effects. Pending I/O must finish during
stopping before this hook runs.
</description>
*)
METHOD PROTECTED OnReset
_RemoveDirectory(bExecute := FALSE);
END_METHOD

(*!
<summary>Validates the configured path and advances the native empty-directory removal request.</summary>
<description>
Computed diagnostic strings are held in local buffers for the duration of the receiving call without dynamic
string-builder allocations.
</description>
*)
METHOD PROTECTED OnRunning
VAR_OUTPUT
	processingState : TOF_Tasks.TASK_PROCESSING_STATE;
END_VAR
VAR_IN_OUT
	stopReasonMessage : TOF_Core.ERROR_MESSAGE;
END_VAR
VAR	
	pathErrorMessage : WSTRING(255);
	formattedExceptionMessage : TOF_Core.ERROR_MESSAGE;
END_VAR
IF NOT _RemoveDirectory.bExecute THEN 
	IF TOF_Core.Strings.IsNullOrWhiteSpace(stringToCheck := _RemoveDirectory.sPathName) THEN
		TOF_Core.Exceptions.ThrowDataMemberNotSpecified(
			sourceNamespaceName := NamespaceName,
			sourceClassName := ClassName,
			sourcePOUName := __POUNAME(),
			sourcePosition := __POSITION(),
			dataMemberName := 'DirectoryPath'
		);		
	END_IF
	
	IF NOT PathHelper.IsValidDirectoryPath(directoryPath := _RemoveDirectory.sPathName, errorMessage => pathErrorMessage) THEN
		FileSystemExceptions.ThrowInvalidPath(
			sourceNamespaceName := NamespaceName,
			sourceClassName := ClassName,
			sourcePOUName := __POUNAME(),
			sourcePosition := __POSITION(),
			path := _RemoveDirectory.sPathName,
			errorMessage := pathErrorMessage
		);
	END_IF
END_IF

_RemoveDirectory(bExecute := TRUE);

IF _RemoveDirectory.bError THEN
	TOF_Core.WideStrings.Append255(
		formattedExceptionMessage,
		"An while removing directory '",
		TO_WSTRING(_RemoveDirectory.sPathName),
		"'");

	FileSystemExceptions.ThrowFileSystem(
		sourceNamespaceName := NamespaceName,
		sourceClassName := ClassName,
		sourcePOUName := __POUNAME(),
		sourcePosition := __POSITION(),
		message := formattedExceptionMessage,
		errorCode := _RemoveDirectory.nErrId
	);
END_IF

IF NOT _RemoveDirectory.bBusy THEN
	processingState := TOF_Tasks.TASK_PROCESSING_STATE.DONE;
END_IF
END_METHOD

(*!
<summary>Waits for an already submitted operation before task termination.</summary>
<description>
Runs for every stop reason. Advances the pending FB with bExecute=FALSE without issuing another request.
Completion does not roll back side effects. Keep configuration and borrowed buffers valid until STOPPED.
</description>
<param name="readyToRelease">TRUE when the underlying FB is no longer busy.</param>
*)
METHOD PROTECTED OnStopping
VAR_OUTPUT
	readyToRelease : BOOL;
END_VAR
IF _RemoveDirectory.bBusy THEN
	_RemoveDirectory(bExecute := FALSE);
END_IF

readyToRelease := NOT _RemoveDirectory.bBusy;
END_METHOD

(*!
<summary>Selects the native path context for the filesystem request.</summary>
<description>
Configure before Start and keep unchanged until STOPPED. It is passed to the native operation, not used as a
path-validity result. Reset preserves it.
</description>
*)
{attribute 'monitoring' := 'call'}
PROPERTY PathType : Tc2_System.E_OpenPath
GET
PathType := _RemoveDirectory.ePath;
END_GET
SET
_RemoveDirectory.ePath := PathType;
END_SET
END_PROPERTY

(*!
<summary>Reports the size of this concrete instance in bytes.</summary>
*)
{attribute 'monitoring' := 'call'}
PROPERTY SelfSize : ULINT
GET
SelfSize := XSIZEOF(THIS^);
END_GET
END_PROPERTY

(*!
<summary>Configures the timeout passed to native operation requests.</summary>
<description>
Set before Start and keep unchanged until STOPPED. Reset preserves this value. It is not an overall task
deadline or a guarantee of resource release after a timeout.
</description>
*)
{attribute 'monitoring' := 'call'}
PROPERTY Timeout : TIME
GET
Timeout := _RemoveDirectory.tTimeout;
END_GET
SET
_RemoveDirectory.tTimeout := Timeout;
END_SET
END_PROPERTY

END_FUNCTION_BLOCK

// ---- Tasks/Directory/CheckDirectoryExists.TcPOU
(*
SPDX-FileCopyrightText: © 2026 Oleksandr Tiutyk <trofimich@gmail.com>
SPDX-License-Identifier: MIT
License: https://opensource.org/license/mit
*)

(*!
<summary>Checks whether a filesystem directory exists through cyclic task execution.</summary>
<description>
Stopping closes an unfinished native enumeration before reporting completion. Diagnostic string inputs are
borrowed only during the call; retained diagnostic text is copied into owned storage. A found file is a
successful check with DirectoryExists=FALSE.
</description>
*)

{attribute 'no_explicit_call' := 'do not call this function block directly'}
FUNCTION_BLOCK CheckDirectoryExists EXTENDS TOF_Tasks.Task IMPLEMENTS IFileSystemTask
VAR_STAT
	//! <summary>Static type metadata available before the base task initializes its default name.</summary>
	{attribute 'hide'}
	_ClassName : STRING := __POUNAME();
END_VAR
VAR
	_EnumFindFile : Tc2_Utilities.FB_EnumFindFileEntry;
	//! <summary>Records whether a search command may still own native enumeration resources.</summary>
	_EnumerationStarted : BOOL;
	//! <summary>Prevents repeating the abort command while its completion is pending.</summary>
	_EnumerationAbortIssued : BOOL;
	
	_DirectoryExists : BOOL;
END_VAR

(*!
<summary>Selects the ADS target for the native filesystem operation.</summary>
<description>
Configure before Start and keep unchanged until STOPPED; the setter stores configuration without submitting
I/O.
</description>
*)
{attribute 'monitoring' := 'call'}
PROPERTY AmsNetId : Tc2_System.T_AmsNetID
GET
AmsNetId := _EnumFindFile.sNetId;
END_GET
SET
_EnumFindFile.sNetId := AmsNetId;
END_SET
END_PROPERTY

(*!
<summary>Provides the concrete type name used in diagnostics.</summary>
<description>
Returns borrowed read-only metadata; keep the instance alive and do not modify the referenced string.
Initialized static storage is ready during base Task.FB_init; this getter has no side effects or exceptions.
</description>
*)
{attribute 'monitoring' := 'call'}
PROPERTY ClassName : REFERENCE TO STRING
GET
ClassName REF= _ClassName;
END_GET
END_PROPERTY

(*!
<summary>Reports whether the completed check found a directory.</summary>
<description>
Meaningful after successful task completion. FALSE means no entry or a found file; a failed search must be
distinguished through FinalStopReason. Reset clears this result.
</description>
*)
{attribute 'monitoring' := 'call'}
PROPERTY DirectoryExists : BOOL
GET
DirectoryExists := _DirectoryExists;
END_GET
END_PROPERTY

(*!
<summary>Provides the copied directory path used by the operation and its existence check.</summary>
<description>
Configure before Start and keep unchanged until STOPPED. PathHelper applies its limited lexical filter before
native submission. Assignment does not perform I/O; Reset preserves the path.
</description>
*)
{attribute 'monitoring' := 'call'}
PROPERTY DirectoryPath : Tc2_System.T_MaxString
GET
DirectoryPath := _EnumFindFile.sPathName;
END_GET
SET
_EnumFindFile.sPathName := DirectoryPath;
END_SET
END_PROPERTY

(*!
<summary>Provides the library namespace used in diagnostics.</summary>
<description>Returns borrowed read-only namespace storage; do not modify the referenced string.</description>
*)
{attribute 'monitoring' := 'call'}
PROPERTY NamespaceName : REFERENCE TO STRING
GET
NamespaceName REF= CurrentNamespace.Name;
END_GET
END_PROPERTY

(*!
<summary>Clears the completed search and its per-run cleanup state for reuse.</summary>
<description>Called only after stopping has completed; it does not abandon a pending enumeration command.</description>
*)
METHOD PROTECTED OnReset
_EnumFindFile(bExecute := FALSE);

_EnumerationStarted := FALSE;
_EnumerationAbortIssued := FALSE;
_DirectoryExists := FALSE;
END_METHOD

(*!
<summary>Checks one directory search and reports whether the found entry is a directory.</summary>
<description>
Starts the search once, then advances it until an entry, end-of-enumeration or error is reported. A found file
leaves DirectoryExists=FALSE and completes successfully. Early completion leaves native enumeration cleanup to
OnStopping. Computed diagnostics are held in local buffers for the duration of the receiving call without
dynamic string-builder allocations.
</description>
<param name="processingState">DONE after a completed search; BUSY while the command is pending.</param>
<param name="stopReasonMessage">Not changed; exceptions provide search failure diagnostics.</param>
*)
METHOD PROTECTED OnRunning
VAR_OUTPUT
	processingState : TOF_Tasks.TASK_PROCESSING_STATE;
END_VAR
VAR_IN_OUT
	stopReasonMessage : TOF_Core.ERROR_MESSAGE;
END_VAR
VAR	
	pathErrorMessage : WSTRING(255);
	formattedExceptionMessage : TOF_Core.ERROR_MESSAGE;
END_VAR
IF NOT _EnumFindFile.bExecute THEN 
	IF TOF_Core.Strings.IsNullOrWhiteSpace(stringToCheck := _EnumFindFile.sPathName) THEN
		TOF_Core.Exceptions.ThrowDataMemberNotSpecified(
			sourceNamespaceName := NamespaceName,
			sourceClassName := ClassName,
			sourcePOUName := __POUNAME(),
			sourcePosition := __POSITION(),
			dataMemberName := 'DirectoryPath'
		);		
	END_IF
	
	IF NOT PathHelper.IsValidDirectoryPath(directoryPath := _EnumFindFile.sPathName, errorMessage => pathErrorMessage) THEN
		FileSystemExceptions.ThrowInvalidPath(
			sourceNamespaceName := NamespaceName,
			sourceClassName := ClassName,
			sourcePOUName := __POUNAME(),
			sourcePosition := __POSITION(),
			path := _EnumFindFile.sPathName,
			errorMessage := pathErrorMessage
		);
	END_IF
	
	_EnumFindFile.eCmd := Tc2_Utilities.E_EnumCmdType.eEnumCmd_First;
END_IF

_EnumerationStarted := TRUE;
_EnumFindFile(bExecute := TRUE);

IF _EnumFindFile.bError THEN
	TOF_Core.WideStrings.Append255(
		formattedExceptionMessage,
		"Error while checking directory '",
		TO_WSTRING(_EnumFindFile.sPathName),
		"'");

	FileSystemExceptions.ThrowFileSystem(
		sourceNamespaceName := NamespaceName,
		sourceClassName := ClassName,
		sourcePOUName := __POUNAME(),
		sourcePosition := __POSITION(),
		message := formattedExceptionMessage,
		errorCode := _EnumFindFile.nErrId
	);
ELSIF NOT _EnumFindFile.bBusy THEN	
	IF NOT _EnumFindFile.bEOE THEN
		_DirectoryExists := _EnumFindFile.stFindFile.fileAttributes.bDirectory;		
	END_IF

	processingState := TOF_Tasks.TASK_PROCESSING_STATE.DONE;
END_IF
END_METHOD

(*!
<summary>Advances directory stop actions before reporting termination.</summary>
<description>
Used for every stop reason. Drains a pending search before deciding whether its native enumeration must be
aborted. An unfinished search receives one abort command with a rising bExecute edge; readiness waits for that
command to complete. End-of-enumeration and search errors need no explicit abort. No new search starts. An
abort error is logged once with its native code and path, without retrying abort or replacing the task stop
reason. Readiness means this cleanup attempt ended, not that server resources were proven released. The log
attempt is made after clearing pending enumeration state; logger failure does not restart cleanup.
</description>
<param name="readyToRelease">TRUE when the directory FBs have finished their pending requests.</param>
*)
METHOD PROTECTED OnStopping
VAR_OUTPUT
	readyToRelease : BOOL;
END_VAR
VAR
	enumerationAbortMessage : WSTRING(255);
END_VAR
IF _EnumerationStarted THEN
	_EnumFindFile(bExecute := FALSE);

	IF NOT _EnumFindFile.bBusy THEN
		IF _EnumFindFile.bEOE OR_ELSE _EnumFindFile.bError THEN
			_EnumerationStarted := FALSE;

			(* End this attempt before reporting its error so logging cannot cause repeated aborts. *)
			IF _EnumerationAbortIssued AND_THEN _EnumFindFile.bError THEN
				enumerationAbortMessage := TOF_Core.WideStrings.Concat255(
					"Directory enumeration abort failed (native error code ",
					TO_WSTRING(_EnumFindFile.nErrId),
					"): ",
					TO_WSTRING(_EnumFindFile.sPathName)
				);
				TOF_Core.LogManager.TryLogMessage(
					message := enumerationAbortMessage,
					category := TOF_Core.LOG_CATEGORY.ERROR,
					topic1 := TO_WSTRING(__POUNAME())
				);
			END_IF
		ELSIF NOT _EnumerationAbortIssued THEN
			_EnumFindFile(bExecute := TRUE, eCmd := Tc2_Utilities.E_EnumCmdType.eEnumCmd_Abort);
			_EnumerationAbortIssued := TRUE;
		ELSE
			_EnumerationStarted := FALSE;
		END_IF
	END_IF
END_IF

readyToRelease := NOT _EnumerationStarted;
END_METHOD

(*!
<summary>Selects the native path context for the filesystem request.</summary>
<description>
Configure before Start and keep unchanged until STOPPED. It is passed to the native operation, not used as a
path-validity result. Reset preserves it. Target support includes the ePath enumeration input in
Tc2_Utilities 3.10.9.
</description>
*)
{attribute 'monitoring' := 'call'}
PROPERTY PathType : Tc2_System.E_OpenPath
GET
PathType := _EnumFindFile.ePath;
END_GET
SET
_EnumFindFile.ePath := PathType;
END_SET
END_PROPERTY

(*!
<summary>Reports the size of this concrete instance in bytes.</summary>
*)
{attribute 'monitoring' := 'call'}
PROPERTY SelfSize : ULINT
GET
SelfSize := XSIZEOF(THIS^);
END_GET
END_PROPERTY

(*!
<summary>Configures the timeout passed to native operation requests.</summary>
<description>
Set before Start and keep unchanged until STOPPED. Reset preserves this value. It is not an overall task
deadline or a guarantee of resource release after a timeout.
</description>
*)
{attribute 'monitoring' := 'call'}
PROPERTY Timeout : TIME
GET
Timeout := _EnumFindFile.tTimeout;
END_GET
SET
_EnumFindFile.tTimeout := Timeout;
END_SET
END_PROPERTY

END_FUNCTION_BLOCK

// ---- Tasks/File/DeleteFile.TcPOU
(*
SPDX-FileCopyrightText: © 2026 Oleksandr Tiutyk <trofimich@gmail.com>
SPDX-License-Identifier: MIT
License: https://opensource.org/license/mit
*)

(*!
<summary>Deletes a file through cyclic task execution.</summary>
<description>
Use one owner task. Configure the path, target, path type and timeout before Start and keep them unchanged
until STOPPED. A missing path is rejected during execution; native errors propagate through Task failure
handling. There is no separate existence check and no conversion of a native not-found error to success.
Continue Execute through stopping, including after cancellation: an already submitted request is drained, not
rolled back. Failure or cancellation does not prove the file still exists. Reset preserves configuration.
</description>
*)

{attribute 'no_explicit_call' := 'do not call this function block directly'}
FUNCTION_BLOCK DeleteFile EXTENDS TOF_Tasks.Task IMPLEMENTS IFileSystemTask
VAR_STAT
	//! <summary>Static type metadata available before the base task initializes its default name.</summary>
	{attribute 'hide'}
	_ClassName : STRING := __POUNAME();
END_VAR
VAR
    _DeleteFile : Tc2_System.FB_FileDelete;
END_VAR

(*!
<summary>Selects the ADS target for the native filesystem operation.</summary>
<description>
Configure before Start and keep unchanged until STOPPED; the setter stores configuration without submitting
I/O.
</description>
*)
{attribute 'monitoring' := 'call'}
{attribute 'OPC.UA.DA.Property' := '1'}
{attribute 'OPC.UA.DA' := '1'}
PROPERTY AmsNetId : Tc2_System.T_AmsNetID
GET
AmsNetId := _DeleteFile.sNetId;
END_GET
SET
_DeleteFile.sNetId := AmsNetId;
END_SET
END_PROPERTY

(*!
<summary>Provides the concrete type name used in diagnostics.</summary>
<description>
Returns borrowed read-only metadata; keep the instance alive and do not modify the referenced string.
Initialized static storage is ready during base Task.FB_init; this getter has no side effects or exceptions.
</description>
*)
{attribute 'monitoring' := 'call'}
PROPERTY ClassName : REFERENCE TO STRING
GET
ClassName REF= _ClassName;
END_GET
END_PROPERTY

(*!
<summary>Provides the configured path for the file operation.</summary>
<description>
The setter copies text without performing I/O. Configure before Start and keep unchanged until STOPPED; Reset
preserves it. The native service determines whether the path is usable.
</description>
*)
{attribute 'monitoring' := 'call'}
{attribute 'OPC.UA.DA.Property' := '1'}
{attribute 'OPC.UA.DA' := '1'}
PROPERTY FilePath : Tc2_System.T_MaxString
GET
FilePath := _DeleteFile.sPathName;
END_GET
SET
_DeleteFile.sPathName := FilePath;
END_SET
END_PROPERTY

(*!
<summary>Provides the library namespace used in diagnostics.</summary>
<description>Returns borrowed read-only namespace storage; do not modify the referenced string.</description>
*)
{attribute 'monitoring' := 'call'}
PROPERTY NamespaceName : REFERENCE TO STRING
GET
NamespaceName REF= CurrentNamespace.Name;
END_GET
END_PROPERTY

(*!
<summary>Resets the native request edge after the task has stopped.</summary>
<description>
Preserves configured inputs and does not undo completed filesystem effects. Pending I/O must finish during
stopping before this hook runs.
</description>
*)
METHOD PROTECTED OnReset
_DeleteFile(bExecute := FALSE);
END_METHOD

(*!
<summary>Submits and advances native deletion of the configured file.</summary>
<description>
Validates required configuration before submitting the request. Native errors raise an exception for the base
Task failure/stopping path without dynamic string-builder allocations. Normal completion reports DONE only
after the native block is no longer busy. No rollback is performed.
</description>
<param name="processingState">BUSY while pending; DONE after native completion without an error.</param>
<param name="stopReasonMessage">Not changed here; failures are passed through exceptions.</param>
*)
METHOD PROTECTED OnRunning
VAR_OUTPUT
	processingState : TOF_Tasks.TASK_PROCESSING_STATE;
END_VAR
VAR_IN_OUT
	stopReasonMessage : TOF_Core.ERROR_MESSAGE;
END_VAR
VAR
	formattedExceptionMessage : TOF_Core.ERROR_MESSAGE;
END_VAR
IF NOT _DeleteFile.bExecute THEN 
	IF TOF_Core.Strings.IsNullOrWhiteSpace(stringToCheck := _DeleteFile.sPathName) THEN
		TOF_Core.Exceptions.ThrowDataMemberNotSpecified(
			sourceNamespaceName := NamespaceName,
			sourceClassName := ClassName,
			sourcePOUName := __POUNAME(),
			sourcePosition := __POSITION(),
			dataMemberName := 'FilePath'
		);		
	END_IF
END_IF

_DeleteFile(bExecute := TRUE);

IF _DeleteFile.bError THEN
	TOF_Core.WideStrings.Append255(
		formattedExceptionMessage,
		"An error occurred while deleting the file '",
		TO_WSTRING(_DeleteFile.sPathName),
		"'");

	FileSystemExceptions.ThrowFileSystem(
		sourceNamespaceName := NamespaceName,
		sourceClassName := ClassName,
		sourcePOUName := __POUNAME(),
		sourcePosition := __POSITION(),
		message := formattedExceptionMessage,
		errorCode := _DeleteFile.nErrId
	);
END_IF

IF NOT _DeleteFile.bBusy THEN
	processingState := TOF_Tasks.TASK_PROCESSING_STATE.DONE;
END_IF
END_METHOD

(*!
<summary>Waits for an already submitted operation before task termination.</summary>
<description>
Runs for every stop reason. Advances the pending FB with bExecute=FALSE without issuing another request.
Completion does not roll back side effects. Keep configuration and borrowed buffers valid until STOPPED.
</description>
<param name="readyToRelease">TRUE when the underlying FB is no longer busy.</param>
*)
METHOD PROTECTED OnStopping
VAR_OUTPUT
	readyToRelease : BOOL;
END_VAR
IF _DeleteFile.bBusy THEN
	_DeleteFile(bExecute := FALSE);
END_IF

readyToRelease := NOT _DeleteFile.bBusy;
END_METHOD

(*!
<summary>Selects the native path context for the filesystem request.</summary>
<description>
Configure before Start and keep unchanged until STOPPED. It is passed to the native operation, not used as a
path-validity result. Reset preserves it.
</description>
*)
{attribute 'monitoring' := 'call'}
{attribute 'OPC.UA.DA.Property' := '1'}
{attribute 'OPC.UA.DA' := '1'}
PROPERTY PathType : Tc2_System.E_OpenPath
GET
PathType := _DeleteFile.ePath;
END_GET
SET
_DeleteFile.ePath := PathType;
END_SET
END_PROPERTY

(*!
<summary>Reports the size of this concrete instance in bytes.</summary>
*)
{attribute 'monitoring' := 'call'}
PROPERTY SelfSize : ULINT
GET
SelfSize := XSIZEOF(THIS^);
END_GET
END_PROPERTY

(*!
<summary>Configures the timeout passed to native operation requests.</summary>
<description>
Set before Start and keep unchanged until STOPPED. Reset preserves this value. It is not an overall task
deadline or a guarantee of resource release after a timeout.
</description>
*)
{attribute 'monitoring' := 'call'}
{attribute 'OPC.UA.DA.Property' := '1'}
{attribute 'OPC.UA.DA' := '1'}
PROPERTY Timeout : TIME
GET
Timeout := _DeleteFile.tTimeout;
END_GET
SET
_DeleteFile.tTimeout := Timeout;
END_SET
END_PROPERTY

END_FUNCTION_BLOCK

// ---- Tasks/File/FileContent/FileContentManager.TcPOU
(*
SPDX-FileCopyrightText: © 2026 Oleksandr Tiutyk <trofimich@gmail.com>
SPDX-License-Identifier: MIT
License: https://opensource.org/license/mit
*)

(*!
<summary>Runs borrowed file-content tasks sequentially using one managed file resource.</summary>
<description>
Use one owner task; do not drive children independently while queued. DiagnosticLogger also selects the
embedded resource manager's independent diagnostic route; configure it before Start and retain its lifetime.
Child tasks retain their own diagnostic destinations. The manager owns its embedded resource
objects, not the children. Keep each child alive until removed; keep this manager alive while any child or
caller uses a borrowed resource reference. Queue removal does not clear a child's binding. Configure FilePath,
ModeFlags, PathType, AmsNetId and Timeout before Start and keep them unchanged until STOPPED. Advance Execute
through stopping and release. A completed best-effort close attempt does not prove physical close success. An
exposed handle is not an acquisition guard and must not be retained across release. Reset from STOPPED clears
queue entries and FilePath; it does not reset children. Reset in READY is a no-op. A removed STOPPED child can
Reset to clear its binding; a removed READY child must explicitly clear or replace its binding before the old
owner is destroyed. Do not mutate borrowed resource data or close its handle directly. Before online change,
stop producers from enqueueing or starting new work. For a running manager, set StopWhenNoPendingTasks to TRUE
to finish queued work, or request Cancel if abandoning waiting work is acceptable. Continue cyclic Execute
until STOPPED, including child completion and resource release. An idle running manager may still hold an open
file. Online change with a retained handle or pending native operation is unsupported; there is no automatic
guard or active-handle handoff. Cleanup errors require resolution before treating the application as prepared;
STOPPED alone does not prove physical release.
</description>
*)

{attribute 'no_explicit_call' := 'Direct call is not allowed'}
FUNCTION_BLOCK FileContentManager EXTENDS TOF_Tasks.TaskQueue
VAR_STAT
	//! <summary>Static type metadata available before the base task initializes its default name.</summary>
	{attribute 'hide'}
	_ClassName : STRING := __POUNAME();
END_VAR
VAR
	{attribute 'hide'} 
	_FileHandleResourceManager : FileHandleResourceManager;
END_VAR

(*!
<summary>Shared target for open, child operations and close. Configure before Start;</summary>
<description>
keep unchanged until STOPPED. Children obtain this target from their resource.
</description>
*)

{attribute 'monitoring' := 'call'}

PROPERTY AmsNetId : Tc2_System.T_AmsNetID
GET
AmsNetId := _FileHandleResourceManager.AmsNetId;
END_GET
SET
_FileHandleResourceManager.AmsNetId := AmsNetId;
END_SET
END_PROPERTY

(*!
<summary>Provides the concrete type name used in diagnostics.</summary>
<description>
Returns borrowed read-only metadata; keep the instance alive and do not modify the referenced string.
Initialized static storage is ready during base Task.FB_init; this getter has no side effects or exceptions.
</description>
*)
{attribute 'monitoring' := 'call'}
PROPERTY ClassName : REFERENCE TO STRING
GET
ClassName REF= _ClassName;
END_GET
END_PROPERTY

(*!
<summary>Binds a prepared file-content task to this manager and appends it to the queue.</summary>
<description>
The child is borrowed, not cloned or owned. It must be READY, alive, unique in this queue and absent from
every other queue. Do not drive or rebind it independently while queued. Successful return means the child was
appended; execution starts later through the queue. Null raises ArgumentNotSpecifiedException in the caller;
this is not a Task FAILURE result. Binding occurs before queue insertion, so an exception does not guarantee
restoration of the previous binding. A custom SetFileHandleResource may also have partial effects before
throwing. Terminal allocation failure must reach the owner's fatal task boundary. Remove a child from its
previous queue before rebinding. Removing entries does not clear their bindings. Reset this manager before
filling it for reuse from STOPPED; its Reset clears entries, not child state.
</description>
<param name="fileHandleTask">Live, unqueued READY task whose execution is delegated to this queue.</param>
*)
METHOD Enqueue
VAR_INPUT
	fileHandleTask : IFileContentTask;
END_VAR
IF fileHandleTask = 0 THEN
	(* A missing required argument cannot be reported as successful enqueue; the caller handles the exception. *)
	TOF_Core.Exceptions.ThrowArgumentNotSpecified(
		sourceNamespaceName := NamespaceName,
		sourceClassName := ClassName,
		sourcePOUName := __POUNAME(),
		sourcePosition := __POSITION(),
		argumentName := 'fileHandleTask'
	);
END_IF

fileHandleTask.SetFileHandleResource(fileHandleResource := _FileHandleResourceManager.FileHandleResource);
EnqueueTask(task := fileHandleTask);
END_METHOD

(*!
<summary>Exposes the native handle associated with this manager.</summary>
<description>
This observation does not check acquisition or physical close success. Do not close it independently or reuse
a saved value after release; file-content tasks use the manager-owned resource.
</description>
*)
{attribute 'monitoring' := 'call'}
PROPERTY FINAL FileHandle : UINT
GET
FileHandle := _FileHandleResourceManager.FileHandle;
END_GET
END_PROPERTY

{attribute 'monitoring' := 'call'}
(*!
<summary>Provides the path of the file to acquire on the configured target.</summary>
<description>
Set before Start and keep unchanged until STOPPED. The setter copies the text; the native open service
resolves it with PathType. It must refer to the target's local filesystem, not a network share. Reset from
STOPPED clears the path. Path assignment does not open or validate an existing file.
</description>
*)
PROPERTY FilePath : Tc2_System.T_MaxString
GET
FilePath := _FileHandleResourceManager.FilePath;
END_GET
SET
_FileHandleResourceManager.FilePath := FilePath;
END_SET
END_PROPERTY

(*!
<summary>Selects native file access and text or binary mode.</summary>
<description>
Configure before Start and keep unchanged until STOPPED. Choose exactly one of FOPEN_MODEREAD, FOPEN_MODEWRITE
or FOPEN_MODEAPPEND, optionally combine FOPEN_MODEPLUS, and explicitly choose one of FOPEN_MODETEXT or
FOPEN_MODEBINARY. Use Tc2_System constants with OR; incompatible choices are rejected by the native open
operation, not validated by this property. WRITE creates or truncates, READ requires an existing file, and
APPEND writes at the end. Omitting text/binary leaves the choice to the native environment. Reset preserves
these flags.
</description>
*)

{attribute 'monitoring' := 'call'}

PROPERTY ModeFlags : DWORD
GET
ModeFlags := _FileHandleResourceManager.ModeFlags;
END_GET
SET
_FileHandleResourceManager.ModeFlags := ModeFlags;
END_SET
END_PROPERTY

(*!
<summary>Provides the library namespace used in diagnostics.</summary>
<description>Returns borrowed read-only namespace storage; do not modify the referenced string.</description>
*)
{attribute 'monitoring' := 'call'}
PROPERTY NamespaceName : REFERENCE TO STRING
GET
NamespaceName REF= CurrentNamespace.Name;
END_GET
END_PROPERTY

(*!
<summary>Clears queued references and the configured file path on Reset from STOPPED.</summary>
<description>
Preserves the inherited queue reset without resetting or deleting children or clearing their resource
bindings. Other manager configuration remains unchanged. READY Reset does not invoke this hook. Overrides must
preserve both queue reset and path clearing.
</description>
*)
METHOD PROTECTED OnReset
SUPER^.OnReset();

FilePath := '';
END_METHOD

(*!
<summary>Wait for the current child and any pending file-open response before release.</summary>
<description>
Runs for every stop reason. A late handle is retained and closed by the normal resource manager.
</description>
<param name="readyToRelease">TRUE after pending work has completed and release may begin.</param>
*)

METHOD PROTECTED OnStopping
VAR_OUTPUT
	readyToRelease : BOOL;
END_VAR
SUPER^.OnStopping(readyToRelease => readyToRelease);

IF readyToRelease THEN
	readyToRelease := _FileHandleResourceManager.FinishPendingAcquire();
END_IF
END_METHOD

{attribute 'monitoring' := 'call'}
(*!
<summary>Selects the native target path context used when opening FilePath.</summary>
<description>
Configure before Start and keep unchanged until STOPPED. Passed to the native open service; it is not a
path-validity result. Reset preserves it.
</description>
*)
PROPERTY PathType : Tc2_System.E_OpenPath
GET
PathType := _FileHandleResourceManager.PathType;
END_GET
SET
_FileHandleResourceManager.PathType := PathType;
END_SET
END_PROPERTY

(*!
<summary>Exposes the file-resource manager borrowed by this task queue.</summary>
<description>
Keep this FileContentManager alive while using the interface. Use it for resource observations; do not
independently request acquisition or release, execute it, or delete it while the queue owns its lifecycle.
</description>
*)
PROPERTY ResourceManager : TOF_Core.IResourceManager
GET
ResourceManager := _FileHandleResourceManager;
END_GET
END_PROPERTY

(*!
<summary>Reports the size of this concrete instance in bytes.</summary>
*)
{attribute 'monitoring' := 'call'}
PROPERTY SelfSize : ULINT
GET
SelfSize := XSIZEOF(THIS^);
END_GET
END_PROPERTY

{attribute 'monitoring' := 'call'}
(*!
<summary>Sets the native timeout for acquiring and releasing this manager's file.</summary>
<description>
Configure before Start and keep unchanged until STOPPED. Children have their own operation timeouts; this
value is not a deadline for the whole queue or its stopping phase. Reset preserves it.
</description>
*)
PROPERTY Timeout : TIME
GET
Timeout := _FileHandleResourceManager.Timeout;
END_GET
SET
_FileHandleResourceManager.Timeout := Timeout;
END_SET
END_PROPERTY

(*!
<summary>Binds the file-resource diagnostic destination before the manager starts.</summary>
<description>
Preserves inherited start preparation. Copies the borrowed DiagnosticLogger to the embedded resource manager
without logging, I/O or ownership transfer. Keep it alive and stable through release.
</description>
*)
METHOD PROTECTED OnBeforeStart
SUPER^.OnBeforeStart();
_FileHandleResourceManager.DiagnosticLogger := THIS^.DiagnosticLogger;
END_METHOD

END_FUNCTION_BLOCK

// ---- Tasks/File/FileContent/FileHandleResourceManager.TcPOU
(*
SPDX-FileCopyrightText: © 2026 Oleksandr Tiutyk <trofimich@gmail.com>
SPDX-License-Identifier: MIT
License: https://opensource.org/license/mit
*)

(*!
<summary>Manages file opening and best-effort closing for file-content tasks.</summary>
<description>
StartAcquire and StartRelease request one operation; Execute advances it until completion. Configure before
acquisition and keep configuration unchanged until release completes. Do not overlap requests.
FinishPendingAcquire drains a pending open during stopping. Close errors are logged and finish the cleanup
attempt. Normal release must be advanced through Execute before destruction. FB_exit only makes a final
best-effort close request and does not wait for or verify its completion. Before online change, the owner must
finish pending acquisition and release through cyclic execution. No pending native operation or retained open
handle may cross online change; this precondition is not enforced automatically.
</description>
*)

{attribute 'no_explicit_call' := 'Direct call is not allowed'}
FUNCTION_BLOCK INTERNAL FileHandleResourceManager EXTENDS TOF_Core.Object IMPLEMENTS TOF_Core.IResourceManager
VAR_STAT
	//! <summary>Class name shared by all instances of this function block.</summary>
	{attribute 'hide'} 
	_ClassName : STRING := __POUNAME();
END_VAR
VAR
	//! <summary>Optional borrowed route that avoids the owning file logger.</summary>
	_DiagnosticLogger : TOF_Core.ILogger;

	_FileOpen : Tc2_System.FB_FileOpen;
	_FileClose : Tc2_System.FB_FileClose;
	
	_FileHandleAcquired : BOOL;
	_Acquiring : BOOL;
	_Releasing : BOOL;
	
	_FileHandleResource : FileHandleResource(fileOpen := _FileOpen);
END_VAR

(*!
<summary>Selects the ADS target for the native filesystem operation.</summary>
<description>
Shared by open and close. Configure before acquisition and keep unchanged through completed release;
assignment does not submit I/O.
</description>
*)
{attribute 'monitoring' := 'call'}
PROPERTY AmsNetId : Tc2_System.T_AmsNetID
GET
AmsNetId := _FileOpen.sNetId;
END_GET
SET
_FileOpen.sNetId := AmsNetId;
_FileClose.sNetId := AmsNetId;
END_SET
END_PROPERTY

(*!
<summary>Provides the concrete type name used in diagnostics.</summary>
<description>
Returns borrowed read-only metadata; keep the instance alive and do not modify the referenced string.
Reading does not allocate memory, initialize resources or transfer ownership.
</description>
*)
{attribute 'monitoring' := 'call'}
PROPERTY ClassName : REFERENCE TO STRING
GET
ClassName REF= _ClassName;
END_GET
END_PROPERTY

(*!
<summary>Selects an independent borrowed destination for file-resource diagnostics.</summary>
<description>
Zero preserves LogManager topics and routing. A nonzero destination is called directly and must not route
back into the owning file logger. The FileContentManager binds this before acquisition. Keep the destination
alive and unchanged until release finishes; no ownership, configuration or cyclic execution is transferred.
</description>
*)
PROPERTY DiagnosticLogger : TOF_Core.ILogger
GET
DiagnosticLogger := _DiagnosticLogger;
END_GET
SET
_DiagnosticLogger := DiagnosticLogger;
END_SET
END_PROPERTY

(*!
<summary>Advances the requested acquire or release operation; does nothing when idle.</summary>
*)
METHOD Execute
IF _Acquiring THEN
	executeAcquire();
ELSIF _Releasing THEN
	executeRelease();
END_IF
END_METHOD

(*!
<summary>Advances opening of the configured file and reports success through ResourceAcquired.</summary>
*)
METHOD PRIVATE executeAcquire
VAR
	message : TOF_Core.ERROR_MESSAGE;	
END_VAR
_FileOpen(bExecute := TRUE);

IF _FileOpen.bError THEN
	_Acquiring := FALSE;

	TOF_Core.WideStrings.Append255(
		message,
		"Error while open file '",
		TO_WSTRING(_FileOpen.sPathName),
		"'");

	FileSystemExceptions.ThrowFileSystem(
		sourceNamespaceName := NamespaceName,
		sourceClassName := ClassName,
		sourcePOUName := __POUNAME(),
		sourcePosition := __POSITION(),
		message := message,
		errorCode := _FileOpen.nErrId
	);
END_IF

IF NOT _FileOpen.bBusy AND_THEN _FileOpen.hFile > 0 THEN
	_Acquiring := FALSE;
	_FileHandleAcquired := TRUE;

	TOF_Core.WideStrings.Append255(
		message,
		"File '",
		TO_WSTRING(_FileOpen.sPathName),
		"' open");

	tryLogDiagnosticMessage(
		message := message,
		category := TOF_Core.LOG_CATEGORY.INFORMATION,
		topic1 := TO_WSTRING(ClassName),
		topic2 := TO_WSTRING(__POUNAME())
	);
END_IF
END_METHOD

(*!
<summary>Advances best-effort file closing; close errors are logged and the cleanup attempt is completed.</summary>
<description>
After native completion, clears the acquired/releasing flags even on close failure. The error message includes
the native nErrId as a decimal code before the file path. Logging does not retry close or convert the close
error to a new exception. Completed cleanup bookkeeping does not prove physical handle closure; logging
delivery depends on the configured logger.
</description>
*)
METHOD PRIVATE executeRelease
VAR	
	message : TOF_Core.ERROR_MESSAGE;	
END_VAR
IF NOT _FileHandleAcquired THEN
	_Releasing := FALSE;
	_FileOpen(bExecute := FALSE);

	RETURN;
END_IF

_FileClose(hFile := _FileOpen.hFile, bExecute := TRUE);

IF NOT _FileClose.bBusy THEN
	_Releasing := FALSE;
	_FileHandleAcquired := FALSE;

	_FileOpen(bExecute := FALSE);

	IF _FileClose.bError THEN
		TOF_Core.WideStrings.Append255(
			message,
			"Error while closing file (native error code ",
			TO_WSTRING(_FileClose.nErrId),
			"): '",
			TO_WSTRING(_FileOpen.sPathName),
			"'");

